      IF (_MessageLevel > E_MessageType.eMessageError)
      THEN
        _stMsg.eType            := E_MessageType.eMessageInfo;
        _stMsg.eSubdevice       := e_Subdevice.Process_LinkedList_Com_DelHead;
        _stMsg.iErrorNumber     := 0;
        _stMsg.sText            := '';
        _stMsg.sText            := concat(_stMsg.sText, TO_STRING(_eState));
        f_MessageSet(_stMsg);
      END_IF
    END_IF
END_CASE
//-----------------------------------------------------------------------------
//-----------------------------------------------------------------------------

ListDelHead                     := _eState;
END_METHOD

METHOD ListDelTail  : e_progress
VAR_INPUT
  Execute           : BOOL;
END_VAR
VAR_INST
  _ListResult       : ST_PROCESS_LIST_RESULT;
  _nErrorId         : UDINT;
  _eState           : E_PROGRESS;
END_VAR
//-----------------------------------------------------------------------------
IF NOT Execute 
THEN 
	_eState                       := E_PROGRESS.PROGRESS_INIT; 
END_IF 
//-----------------------------------------------------------------------------
IF NOT Check() 
THEN 
	ListDelTail                   := E_PROGRESS.PROGRESS_ERROR; 
	RETURN; 
END_IF
//-----------------------------------------------------------------------------
//-----------------------------------------------------------------------------
CASE _eState
OF
  E_PROGRESS.PROGRESS_INIT:
    IF Execute
    THEN
      _nErrorId                 := 0;
      _eState                   := E_PROGRESS.PROGRESS_BUSY;
    END_IF
END_CASE
//-----------------------------------------------------------------------------
//-----------------------------------------------------------------------------
CASE _eState
OF
  E_PROGRESS.PROGRESS_BUSY:
    _eState                     := E_PROGRESS.PROGRESS_PREPARE;
    _ListResult                 := _ItfList.RemoveTailValue();
END_CASE
//-----------------------------------------------------------------------------
//-----------------------------------------------------------------------------
CASE _eState
OF
  E_PROGRESS.PROGRESS_PREPARE:

    IF (_ListResult.wState <> 0)
    THEN
      _eState                   := E_PROGRESS.PROGRESS_ERROR;
      _nErrorId                 := _ListResult.wState;

      _stMsg.eType              := E_MessageType.eMessageError;
      _stMsg.eSubdevice         := e_Subdevice.Process_LinkedList_Com_DelTail;
      _stMsg.iErrorNumber       := _nErrorId;
      _stMsg.sText              := '';
      _stMsg.sText              := concat(_stMsg.sText, TO_STRING(_eState));
      f_MessageSet(_stMsg);

    ELSE
      _eState                   := E_PROGRESS.PROGRESS_DONE;

      IF (_MessageLevel > E_MessageType.eMessageError)
      THEN
        _stMsg.eType            := E_MessageType.eMessageInfo;
        _stMsg.eSubdevice       := e_Subdevice.Process_LinkedList_Com_DelTail;
        _stMsg.iErrorNumber     := 0;
        _stMsg.sText            := '';
        _stMsg.sText            := concat(_stMsg.sText, TO_STRING(_eState));
        f_MessageSet(_stMsg);
      END_IF
    END_IF
END_CASE
//-----------------------------------------------------------------------------
//-----------------------------------------------------------------------------

ListDelTail                     := _eState;
END_METHOD

METHOD ListGetHead  : e_progress
VAR_INPUT
  Execute           : BOOL;
END_VAR
VAR_INST
  _ListResult       : ST_PROCESS_LIST_RESULT;
  _nErrorId         : UDINT;
  _eState           : E_PROGRESS;
END_VAR
//-----------------------------------------------------------------------------
IF NOT Execute 
THEN 
	_eState                         := E_PROGRESS.PROGRESS_INIT; 
END_IF 
//-----------------------------------------------------------------------------
IF NOT Check() 
THEN 
	ListGetHead                     := E_PROGRESS.PROGRESS_ERROR; 
	RETURN; 
END_IF
//-----------------------------------------------------------------------------
//-----------------------------------------------------------------------------
CASE _eState
OF
  E_PROGRESS.PROGRESS_INIT:
    IF Execute
    THEN
      _nErrorId                   := 0;
      _eState                     := E_PROGRESS.PROGRESS_BUSY;
    END_IF
END_CASE
//-----------------------------------------------------------------------------
//-----------------------------------------------------------------------------
CASE _eState
OF
  E_PROGRESS.PROGRESS_BUSY:
    _eState                       := E_PROGRESS.PROGRESS_PREPARE;
    _ListResult                   := _ItfList.GetHead();
END_CASE
//-----------------------------------------------------------------------------
//-----------------------------------------------------------------------------
CASE _eState
OF
  E_PROGRESS.PROGRESS_PREPARE:

    IF (_ListResult.wState <> 0)
    THEN
      _eState                     := E_PROGRESS.PROGRESS_ERROR;
      _nErrorId                   := _ListResult.wState;

      _stMsg.eType                := E_MessageType.eMessageError;
      _stMsg.eSubdevice           := e_Subdevice.Process_LinkedList_Com_GetHead;
      _stMsg.iErrorNumber         := _nErrorId;
      _stMsg.sText                := '';
      _stMsg.sText                := concat(_stMsg.sText, TO_STRING(_eState));
      f_MessageSet(_stMsg);

    ELSE
      _stNodeDataProcess.ProcessData:= _ListResult.stData;
      _stNodeDataOutput             := _stNodeDataProcess;

      _eState                     := E_PROGRESS.PROGRESS_DONE;

      IF (_MessageLevel > E_MessageType.eMessageError)
      THEN
        _stMsg.eType              := E_MessageType.eMessageInfo;
        _stMsg.eSubdevice         := e_Subdevice.Process_LinkedList_Com_GetHead;
        _stMsg.iErrorNumber       := 0;
        _stMsg.sText              := '';
        _stMsg.sText              := concat(_stMsg.sText, TO_STRING(_eState));
        f_MessageSet(_stMsg);
      END_IF
    END_IF
END_CASE
//-----------------------------------------------------------------------------
//-----------------------------------------------------------------------------

ListGetHead                       := _eState;
END_METHOD

METHOD ListGetTail  : e_progress
VAR_INPUT
  Execute           : BOOL;
END_VAR
VAR_INST
  _ListResult       : ST_PROCESS_LIST_RESULT;
  _nErrorId         : UDINT;
  _eState           : E_PROGRESS;
END_VAR
//-----------------------------------------------------------------------------
IF NOT Execute 
THEN 
	_eState                         := E_PROGRESS.PROGRESS_INIT; 
END_IF 
//-----------------------------------------------------------------------------
IF NOT Check() 
THEN 
	ListGetTail                     := E_PROGRESS.PROGRESS_ERROR; 
	RETURN; 
END_IF
//-----------------------------------------------------------------------------
//-----------------------------------------------------------------------------
CASE _eState
OF
  E_PROGRESS.PROGRESS_INIT:
    IF Execute
    THEN
      _nErrorId                   := 0;
      _eState                     := E_PROGRESS.PROGRESS_BUSY;
    END_IF
END_CASE
//-----------------------------------------------------------------------------
//-----------------------------------------------------------------------------
CASE _eState
OF
  E_PROGRESS.PROGRESS_BUSY:
    _eState                       := E_PROGRESS.PROGRESS_PREPARE;
    _ListResult                   := _ItfList.GetTail();
END_CASE
//-----------------------------------------------------------------------------
//-----------------------------------------------------------------------------
CASE _eState
OF
  E_PROGRESS.PROGRESS_PREPARE:

    IF (_ListResult.wState <> 0)
    THEN
      _eState                     := E_PROGRESS.PROGRESS_ERROR;
      _nErrorId                   := _ListResult.wState;

      _stMsg.eType                := E_MessageType.eMessageError;
      _stMsg.eSubdevice           := e_Subdevice.Process_LinkedList_Com_GetTail;
      _stMsg.iErrorNumber         := _nErrorId;
      _stMsg.sText                := '';
      _stMsg.sText                := concat(_stMsg.sText, TO_STRING(_eState));
      f_MessageSet(_stMsg);

    ELSE
      _stNodeDataProcess.ProcessData:= _ListResult.stData;
      _stNodeDataOutput             := _stNodeDataProcess;

      _eState                     := E_PROGRESS.PROGRESS_DONE;

      IF (_MessageLevel > E_MessageType.eMessageError)
      THEN
        _stMsg.eType              := E_MessageType.eMessageInfo;
        _stMsg.eSubdevice         := e_Subdevice.Process_LinkedList_Com_GetTail;
        _stMsg.iErrorNumber       := 0;
        _stMsg.sText              := '';
        _stMsg.sText              := concat(_stMsg.sText, TO_STRING(_eState));
        f_MessageSet(_stMsg);
      END_IF
    END_IF
END_CASE
//-----------------------------------------------------------------------------
//-----------------------------------------------------------------------------

ListGetTail                       := _eState;
END_METHOD

METHOD ListInit  : e_progress
VAR_INPUT
  Execute           : BOOL;
END_VAR
VAR_INST
  _ListResult       : BOOL;

  _nErrorId         : UDINT;
  _eState           : E_PROGRESS;
END_VAR
//-----------------------------------------------------------------------------
IF NOT Execute 
THEN 
	_eState                       := E_PROGRESS.PROGRESS_INIT; 
END_IF 
//-----------------------------------------------------------------------------
IF NOT Check() 
THEN 
	ListInit                      := E_PROGRESS.PROGRESS_ERROR; 
	RETURN; 
END_IF
//-----------------------------------------------------------------------------
//-----------------------------------------------------------------------------
CASE _eState
OF
  E_PROGRESS.PROGRESS_INIT:
    IF Execute
    THEN
      _nErrorId                 := 0;
      _eState                   := E_PROGRESS.PROGRESS_BUSY;
    END_IF
END_CASE
//-----------------------------------------------------------------------------
//-----------------------------------------------------------------------------
CASE _eState
OF
  E_PROGRESS.PROGRESS_BUSY:
    _eState                     := E_PROGRESS.PROGRESS_PREPARE;
    _ListResult                 := _ItfList.InitList();
END_CASE
//-----------------------------------------------------------------------------
//-----------------------------------------------------------------------------
CASE _eState
OF
  E_PROGRESS.PROGRESS_PREPARE:

    IF NOT (_ListResult)
    THEN
      _eState                   := E_PROGRESS.PROGRESS_ERROR;
      _nErrorId                 := 666;

      _stMsg.eType              := E_MessageType.eMessageError;
      _stMsg.eSubdevice         := e_Subdevice.Process_LinkedList_Com_Init;
      _stMsg.iErrorNumber       := _nErrorId;
      _stMsg.sText              := '';
      _stMsg.sText              := concat(_stMsg.sText, TO_STRING(_eState));
      f_MessageSet(_stMsg);

    ELSE
      _eState                   := E_PROGRESS.PROGRESS_DONE;

      IF (_MessageLevel > E_MessageType.eMessageError)
      THEN
        _stMsg.eType            := E_MessageType.eMessageInfo;
        _stMsg.eSubdevice       := e_Subdevice.Process_LinkedList_Com_Init;
        _stMsg.iErrorNumber     := 0;
        _stMsg.sText            := '';
        _stMsg.sText            := concat(_stMsg.sText, TO_STRING(_eState));
        f_MessageSet(_stMsg);
      END_IF
    END_IF
END_CASE
//-----------------------------------------------------------------------------
//-----------------------------------------------------------------------------

ListInit                        := _eState;
END_METHOD

PROPERTY MessageLevel : e_MessageType
GET
MessageLevel := _MessageLevel;
END_GET
SET
_MessageLevel := MessageLevel;
END_SET
END_PROPERTY

PROPERTY NodeDataInput : reference to st_list_node_data
SET
_stNodeDataInput REF= NodeDataInput;
END_SET
END_PROPERTY

PROPERTY NodeDataOutput : reference to st_list_node_data
SET
_stNodeDataOutput REF= NodeDataOutput;
END_SET
END_PROPERTY

PROPERTY State : REFERENCE TO ST_LIST_STATE
SET
_stState ref= State;
END_SET
END_PROPERTY

END_FUNCTION_BLOCK

// ---- XTS_TRANSPORT/MAIN_XTS.TcPOU
//---------------------------------------------------------------------------------------------------------------
//
//  HAUD 2026.07.25
//  - refactoring update
//    - folder structure accommodates PLC_MOTION_LAYER MSG declarations
//      - This shall help to have both projects merged into one codebase
//        - merging this into a single codebase is up to you, 
//          the machines I do are vastly different in that regard
//          I merge what I need for an implementation / example
//
//    - PRGs are in their corresponding folders
//      - MAIN_XTS --> [XTS]
//      - MAIN_APP --> [APPLICATION]
//
//    - Manage the call tree when merging --> PlcTask.TcTTO
//
//---------------------------------------------------------------------------------------------------------------
//
//  HAUD 2026.07.24
//  - message system refactoring
//    - XTS_TRANSPORT_LAYER and PLC_MOTION_LAYER merged devices
//      - GVL naming conflict resolved
//---------------------------------------------------------------------------------------------------------------
//
//  HAUD 2026.04.23
//  - fb_Xpu
//    - .Init() initialisation sequence with explicit init of all local instances
//    - .GetPartModule added, gets all Tc3_XTS_Utility.I_TcIoXtsPartModule 
// 
//  - MAPPING
//    - MOVER_SELECTOR and MOVER_MAPPING compile defines are mutually exclusive.
//    - switching memcpy destinations/sources according to compile define
//
//  - I_XtsTransport_Xpu
//    - you might need this interface to access methods for passing along the XTS_Utility interfaces
//
// 
//---------------------------------------------------------------------------------------------------------------
//
//  HAUD 2026.03.15
//  - refactoring of the constants
//  - I never really used the parameter list anyway 
//
//  - XTS Utility lib parameter and project constants now reside in:
//    GVL_XTS_CONSTANTS
//
//  - addition of MAIN_APP (also see call tree)
//    - this might be a point of entry for you
//    - advanced transport logic may live here
//    - Beware the Collectors, they need instances to be really useful
//
//---------------------------------------------------------------------------------------------------------------
//
//  HAUD 2026.02.11
//  - transport layer new member:
//    - MoverSelector
//      - Cyclic movement execution class
//      - mapping unions available
//      - Mover selection (one mover at a time)
//      - composition using I_XtsTransport_Mover
//
//
//---------------------------------------------------------------------------------------------------------------
//
//  HAUD 2025.12.04
//
//  - XTS_TRANSPORT_LAYER
//  - transport layer members:
//    - MessageData
//      - ABSTRACT base class
//        - cyclic wrapper
//
//      - device driven message list implementation
//        - e_Device.Metrics: message list dedicated for performance logs
//
//      - new e_MessageType
//        -  eMessageBatch: may be used for performance metric messages
//
//    - CaGroup
//      - access to Group functions
//
//    - Mover
//      - Base class
//        - cyclic wrapper
//
//      - access to MC and CA motion functions
//
//    - Xpu (ProcessingUnit)
//      - Base class
//        - cyclic wrapper
//
//      - access to TcCOM Objects in Environment
//
//    - Transport Control Unit
//      - coordinates members to get XTS in defined states
//
//    - Xts Stations
//      - ABSTRACT base class
//        - used via inheritance
//
//      - handshakes with extern control for mover transport
//
//  - global datafields for mrmbers in GVL_XTS namespace
//  - global interface datafields for use in members
//  - structures are assigned by reference for every member
//
//---------------------------------------------------------------------------------------------------------------
// HAUD 2025 08 29
//
//    XTS_TRANSPORT_LAYER project
//    
//    MIT License
//    
//    Copyright (c) 2025 HAUD
//    
//    Permission is hereby granted, free of charge, to any person obtaining a copy
//    of this software and associated documentation files (the "Software"), to deal
//    in the Software without restriction, including without limitation the rights
//    to use, copy, modify, merge, publish, distribute, sublicense, and/or sell
//    copies of the Software, and to permit persons to whom the Software is
//    furnished to do so, subject to the following conditions:
//    
//    The above copyright notice and this permission notice shall be included in all
//    copies or substantial portions of the Software.
//    
//    THE SOFTWARE IS PROVIDED "AS IS", WITHOUT WARRANTY OF ANY KIND, EXPRESS OR
//    IMPLIED, INCLUDING BUT NOT LIMITED TO THE WARRANTIES OF MERCHANTABILITY,
//    FITNESS FOR A PARTICULAR PURPOSE AND NONINFRINGEMENT. IN NO EVENT SHALL THE
//    AUTHORS OR COPYRIGHT HOLDERS BE LIABLE FOR ANY CLAIM, DAMAGES OR OTHER
//    LIABILITY, WHETHER IN AN ACTION OF CONTRACT, TORT OR OTHERWISE, ARISING FROM,
//    OUT OF OR IN CONNECTION WITH THE SOFTWARE OR THE USE OR OTHER DEALINGS IN THE
//    SOFTWARE.
//---------------------------------------------------------------------------------------------------------------
PROGRAM MAIN_XTS
VAR
  //-------------------------------------------------------------------------------------------------------------
  //  MAIN - important members
  //-------------------------------------------------------------------------------------------------------------
  eInit                   : E_PROGRESS; // startup states
  eInitError              : E_PROGRESS; // startup error state: NOT_EXIST --> NO_ERROR

  nStation,
	nMover                  : UINT;
  //-------------------------------------------------------------------------------------------------------------
  //-------------------------------------------------------------------------------------------------------------
  // default initialization data
  //-------------------------------------------------------------------------------------------------------------
  nStn                    : UINT;               // startup default data, do not delete
  rInitVelo               : REAL :=     500.0;  // default data, use your own in a real machine!
  rInitGap                : REAL :=     100.0;  // default data, use your own in a real machine!
  rInitAcc                : REAL :=  10_000.0;  // default data, use your own in a real machine!
  rInitJerk               : REAL := 100_000.0;  // default data, use your own in a real machine!
  //-------------------------------------------------------------------------------------------------------------
  //-------------------------------------------------------------------------------------------------------------
  // message data used here in MAIN (init state machine etc.)
  //-------------------------------------------------------------------------------------------------------------
  stMsg                   : ST_Message;
  eMsgState               : e_message_state;
  eMsgProgress            : E_PROGRESS;
  eMtrState               : e_message_state;
  eMtrProgress            : E_PROGRESS;
  //-------------------------------------------------------------------------------------------------------------
  //-------------------------------------------------------------------------------------------------------------
  // visualisations - the helper visus depend on these
  //                - the helper visus are just that
  //-------------------------------------------------------------------------------------------------------------
  nMoverSelected,
  nStationSelected,
  nStationParameter       : UINT;

  sStationText            : STRING(30);
  stXpuStrings            : ST_XPU_STRINGS;

  eTransportState         : E_XTS_TRANSPORT_STATE;
  eTransportResult        : E_PROGRESS;

  eXpuState               : E_XPU_STATE;
  eXpuResult              : E_PROGRESS;
  eXpuCheck               : E_XPU_CHECK;

  eSelectorState,
  eMoverState             : E_MOVER_STATE;

  eSelectorResult,
  eMoverResult            : E_PROGRESS;

  sSelectorState,
  sSelectorResult,
  sCaGroupState,
  sTransportState,
  sTransportCheck,
  sTransportResult,
  sMoverState,
  sMoverResult,
  sStationState,
  sStationStateMask,
  sStationCtrlMask        : STRING;

  bStationEnable,
  bStationEnter,
  bStationStart,
  bStationDone,
  bStationOut,
  bStationGone            : BOOL;

  tStationSelectedQueue   : ARRAY[1..MAX_LIST_NODES] OF ST_STATION_MOVER_DATA;
  //-------------------------------------------------------------------------------------------------------------
  tIdleWriteMotion        : TIME := T#5S;
  tIdleWriteMetric        : TIME := T#5S;
  tonIdleWriteMotion      : Tc2_Standard.TON;
  tonIdleWriteMetric      : Tc2_Standard.TON;
  //-------------------------------------------------------------------------------------------------------------
END_VAR

//############################################################################
// Local time; used for timestamps
//############################################################################
GVL_MSG_XTS.fbLocalTime();
GVL_MSG_XTS.sLocalTime                              := GVL_MSG_XTS.fbLocalTime.LocalTimeString;
GVL_MSG_XTS.dtLocalTime                             := GVL_MSG_XTS.fbLocalTime.LocalTime;
//############################################################################
//############################################################################
// 	example for init sequence
//############################################################################	
CASE eInit
OF
  E_PROGRESS.PROGRESS_INVALID:
    // In the beginning there was no error...
    eInitError                                  := E_PROGRESS.PROGRESS_NOT_EXIST;
    //---------------------------------------------------------------------------
    // where are the stations?
    // TODO: after importing this project into your XTS TwinCAT solution
    //       setup of Station parameters is required.
    //---------------------------------------------------------------------------
    // default initialization, please leave this in here
    DefaultStationParameters();        
    //---------------------------------------------------------------------------
    //---------------------------------------------------------------------------
    // where to start?
    // fb_TransportUnit is connected StationStartIndex and StationStart
    //
    // TODO: after importing this project into your XTS TwinCAT solution
    //       setup of StartStation parameters is up to you to decide.
    //---------------------------------------------------------------------------
    GVL_XTS.StationStartIndex                   := 1; // this index is yours to change, fbTransportUnit is connected to it
    GVL_XTS.StationStart                        := GVL_XTS.StationParameter[GVL_XTS.StationStartIndex]; // put in here any plausible data you like
    //---------------------------------------------------------------------------

    eInit                                       := E_PROGRESS.PROGRESS_BUSY;
    // clear command interface
    GVL_XTS.XpuCtrl.Cmd                         := E_XPU_CTRL.XTS_CMD_NULL;
    GVL_MSG_XTS.TransportMessageCtrl.Cmd            := E_MESSAGE_CTRL.MSG_CTRL_NULL;
    GVL_MSG_XTS.MetricsMessageCtrl.Cmd              := E_MESSAGE_CTRL.MSG_CTRL_NULL;

    // set detailed message levvel for startup
    GVL_MSG_XTS.MessageLevelXpu                     := E_MessageType.eMessageVerbose; //GVL_MSG.MessageLevel;
    GVL_XTS.CaGroup.MessageLevel                := E_MessageType.eMessageVerbose; //GVL_MSG.MessageLevel;
    GVL_XTS.XtsTransport.MessageLevel           := E_MessageType.eMessageVerbose; //GVL_MSG.MessageLevel;

    FOR nStation := 1 TO MAX_STATION
    DO
      GVL_MSG_XTS.MessageLevelStations[nStation]    := E_MessageType.eMessageVerbose; //GVL_MSG.MessageLevel;
    END_FOR
    FOR nMover := 1 TO MAX_MOVER
    DO
      GVL_MSG_XTS.MessageLevelMovers[nMover]        := E_MessageType.eMessageVerbose; //GVL_MSG.MessageLevel;
    END_FOR
    
  //-----------------------------------------------------------------------------
  //-----------------------------------------------------------------------------
  E_PROGRESS.PROGRESS_BUSY:         // init Xpu, ProcessingUnit, MotorModules
    eInit                                       := E_PROGRESS.PROGRESS_PREPARE;
    GVL_MSG_XTS.TransportMessageCtrl.Cmd            := E_MESSAGE_CTRL.MSG_CTRL_INIT;
    GVL_MSG_XTS.MetricsMessageCtrl.Cmd              := E_MESSAGE_CTRL.MSG_CTRL_INIT;


  //-----------------------------------------------------------------------------
  //-----------------------------------------------------------------------------
  E_PROGRESS.PROGRESS_PREPARE:      // wait for init to be done
    GVL_XTS.XpuCtrl.Cmd                         := E_XPU_CTRL.XTS_CMD_INIT;
    IF (GVL_XTS.XpuState.State      = E_XPU_STATE.XTS_INIT + E_PROGRESS.PROGRESS_ERROR)
    THEN
      stMsg.eType                               := E_MessageType.eMessageInfo;
      stMsg.eDevice                             := e_Device.Device_Main;
      stMsg.eSubdevice                          := e_Subdevice.MainInit;
      stMsg.iErrorNumber                        := GVL_XTS.XpuState.Check;
      stMsg.sText                               := concat('MAIN.eInit Error: ', TO_STRING(MAIN_XTS.eInit));
      stMsg.sText                               := concat(stMsg.sText , ': ');
      stMsg.sText                               := concat(stMsg.sText, 'XpuState.Check: ');
      stMsg.sText                               := concat(stMsg.sText, TO_STRING(GVL_XTS.XpuState.Check));
      f_MessageSet(stMsg);

      eInitError                                := eInit;
      eInit                                     := E_PROGRESS.PROGRESS_ERROR;

    ELSIF (GVL_XTS.XpuState.State   = E_XPU_STATE.XTS_INIT + E_PROGRESS.PROGRESS_DONE)
    THEN
      eInit                                     := E_PROGRESS.PROGRESS_STARTUP;
      GVL_XTS.XpuCtrl.Cmd                       := E_XPU_CTRL.XTS_IDLE;
    END_IF

  //-----------------------------------------------------------------------------
  //-----------------------------------------------------------------------------
  E_PROGRESS.PROGRESS_STARTUP:
    CASE GVL_XTS.XpuState.Check
    OF
      E_XPU_CHECK.MOVER_ID_SIMULATION,
      E_XPU_CHECK.MOVER_ID_DETECTION_VALID:
        IF (GVL_XTS.XpuState.State = E_XPU_STATE.XTS_IDLE + E_PROGRESS.PROGRESS_WORKING)
        THEN
          eInit                                     := E_PROGRESS.PROGRESS_CHECK;
        END_IF
    END_CASE
  //-----------------------------------------------------------------------------
  //-----------------------------------------------------------------------------
  E_PROGRESS.PROGRESS_CHECK:
    eInit                                       := E_PROGRESS.PROGRESS_OCCUPIED;

  //-----------------------------------------------------------------------------
  //-----------------------------------------------------------------------------
  E_PROGRESS.PROGRESS_OCCUPIED:
    //---------------------------------------------------------------------------
    // how many nests to start with?
    // - this is for you to decide and me to secure, 
    //    so leave the initialisation as it is
    //
    // TODO: after importing this project into your XTS TwinCAT solution
    //       setup of StartStation NestMask configuration is up to you to decide.
    //---------------------------------------------------------------------------
    IF (GVL_XTS.XtsTransport.StationStartIndex > 0) AND
       (GVL_XTS.XtsTransport.StationStartIndex < MAX_STATION+1)
    THEN
      GVL_XTS.StationStart.nConfiguredStopCount := GVL_XTS.StationParameter[GVL_XTS.XtsTransport.StationStartIndex].nConfiguredStopCount;
    END_IF
    eInit                                       := E_PROGRESS.PROGRESS_WORKING;

  //-----------------------------------------------------------------------------
  //-----------------------------------------------------------------------------
  E_PROGRESS.PROGRESS_WORKING:
    GVL_MSG_XTS.TransportMessageCtrl.Cmd            := E_MESSAGE_CTRL.MSG_CTRL_WRITE;
    eInit                                       := E_PROGRESS.PROGRESS_DONE;

    stMsg.eType                                 := E_MessageType.eMessageInfo;
    stMsg.eDevice                               := e_Device.Device_Main;
    stMsg.eSubdevice                            := e_Subdevice.MainInit;
    stMsg.iErrorNumber                          := GVL_XTS.XpuState.Check;
    stMsg.sText                                 := concat('MAIN.eInit Done: ', TO_STRING(MAIN_XTS.eInit));
    stMsg.sText                                 := concat(stMsg.sText , ': ');
    stMsg.sText                                 := concat(stMsg.sText, 'XpuState.Check: ');
    stMsg.sText                                 := concat(stMsg.sText, TO_STRING(GVL_XTS.XpuState.Check));
    f_MessageSet(stMsg);

    //---------------------------------------------------------------------------
END_CASE
//############################################################################
//############################################################################
// 	/XTS Transport Unit
//############################################################################
//  - main control function block for transport layer
//  - requires access to member controls
//    - Xpu
//    - CaGroup
//    - Mover
//    - Station Control
//    - Station LinkedList Interface
//############################################################################
//
// cyclic call
GVL_XTS.XtsTransport();

// main control
GVL_XTS.XtsTransport.Ctrl                       REF= GVL_XTS.XtsTransportCtrl;   // main control
GVL_XTS.XtsTransport.State                      REF= GVL_XTS.XtsTransportState;  // main state
                                        
// member controls                      
GVL_XTS.XtsTransport.XpuCtrl                    REF= GVL_XTS.XpuCtrl;
GVL_XTS.XtsTransport.XpuState                   REF= GVL_XTS.XpuState;
GVL_XTS.XtsTransport.XpuInfo                    REF= GVL_XTS.XpuInfo;
                                        
GVL_XTS.XtsTransport.GroupItf                   :=   GVL_XTS.CaGroupItf;
GVL_XTS.XtsTransport.GroupInfo                  REF= GVL_XTS.CaGroupInfo;
                                        
GVL_XTS.XtsTransport.MoverItf                   REF= GVL_XTS.MoverItf;
GVL_XTS.XtsTransport.MoverInfo                  REF= GVL_XTS.MoverInfo;
GVL_XTS.XtsTransport.MoverLastPosition          REF= GVL_XTS.LastPosition;
GVL_XTS.XtsTransport.MoverLastGap               REF= GVL_XTS.LastGap;

GVL_XTS.XtsTransport.StationStartIndex          :=   GVL_XTS.StationStartIndex;                                        
GVL_XTS.XtsTransport.StationStart               REF= GVL_XTS.StationStart;      // start position for E_XTS_TRANSPORT_CTRL.CMD_TRANSPORT_START
GVL_XTS.XtsTransport.StationCtrlItf             REF= GVL_XTS.StationCtrlItf;    // station interfaces are required for accessing station methods
GVL_XTS.XtsTransport.StationListsItf            REF= GVL_XTS.StationListItf;    // list interface is required for access to linked list methods
GVL_XTS.XtsTransport.StationControl             REF= GVL_XTS.StationCtrl;
GVL_XTS.XtsTransport.StationState               REF= GVL_XTS.StationState;
//############################################################################
// 	XTS Transport Unit/
//############################################################################
//############################################################################
//############################################################################
// 	/XTS Stations
//############################################################################	
FOR nStation := 1 TO MAX_STATION
DO
  // epimetheus assembles the body
  GVL_XTS.StationListItf[nStation]              := GVL_XTS.StationList[nStation];   // interfaces for list methods
  GVL_XTS.StationCtrlItf[nStation]              := GVL_XTS.Station[nStation];       // interfaces for station methods

  CASE GVL_XTS.StationParameter[nStation].eType
  OF
    //-----------------------------------------------------------------------------
    E_STATION_TYPE.STATION_PROCESS:
      GVL_XTS.Station[nStation].MessageLevel    := GVL_MSG_XTS.MessageLevelStations[nStation];

      GVL_XTS.Station[nStation].StationId       := nStation;  // Know Thyself!

    
      GVL_XTS.Station[nStation].Ctrl            REF= GVL_XTS.StationCtrl;           // station ctrl from extern
      GVL_XTS.Station[nStation].State           REF= GVL_XTS.StationState;          // station state to extern
    
      GVL_XTS.Station[nStation].ItfStations     REF= GVL_XTS.StationListItf;        // give every station all list interfaces for writing mover tickets
      GVL_XTS.Station[nStation].ItfMover        REF= GVL_XTS.MoverItf;              // give every station all mover interfaces for movement in / out of station
      GVL_XTS.Station[nStation].Mover           REF= GVL_XTS.AxisRefMover;          // AXIS_REF to read infos from
      GVL_XTS.Station[nStation].MoverOffset     REF= GVL_XTS.PositionOffset;        // static offsets for all stations, all movers, all stop positions
    
      GVL_XTS.Station[nStation].StationParameter  REF= GVL_XTS.StationParameter;// give every station all station parameters for sending to WaitPos of target station
    
      // cyclic call
      GVL_XTS.Station[nStation].Cycle();                                        // cycle for handshaking with extern
    
      // Queue data for each station
      GVL_XTS.StationQueue[nStation]            := GVL_XTS.StationListItf[nStation].Data;


    //-----------------------------------------------------------------------------
    E_STATION_TYPE.STATION_GEAR_IN_POS:
      GVL_XTS.StationGearIn[nStation].MessageLevel:= GVL_MSG_XTS.MessageLevelStations[nStation];

      GVL_XTS.Station[nStation].StationId         := nStation;  // Know Thyself!
    
      GVL_XTS.StationGearIn[nStation].Ctrl        REF= GVL_XTS.StationCtrl;           // station ctrl from extern
      GVL_XTS.StationGearIn[nStation].State       REF= GVL_XTS.StationState;          // station state to extern
    
      GVL_XTS.StationGearIn[nStation].ItfStations REF= GVL_XTS.StationListItf;        // give every station all list interfaces for writing mover tickets
      GVL_XTS.StationGearIn[nStation].ItfMover    REF= GVL_XTS.MoverItf;              // give every station all mover interfaces for movement in / out of station
      GVL_XTS.StationGearIn[nStation].Mover       REF= GVL_XTS.AxisRefMover;          // AXIS_REF to read infos from
      GVL_XTS.StationGearIn[nStation].MoverOffset REF= GVL_XTS.PositionOffset;        // static offsets for all stations, all movers, all stop positions
    
    
      GVL_XTS.StationGearIn[nStation].StationParameter  REF= GVL_XTS.StationParameter;// give every station all station parameters for sending to WaitPos of target station
    
      // cyclic call
      GVL_XTS.StationGearIn[nStation].Cycle();                                        // cycle for handshaking with extern
    
      // Queue data for each station
      GVL_XTS.StationQueue[nStation]            := GVL_XTS.StationListItf[nStation].Data;
  ELSE
      //---------------------------------------------------------------------------------
      // no valid station type --> no identity
      //---------------------------------------------------------------------------------
      GVL_XTS.Station[nStation].StationId       := 0; // I am no one
      //---------------------------------------------------------------------------------
  END_CASE
END_FOR
//############################################################################
// 	XTS Stations/
//############################################################################	
//############################################################################
//############################################################################
// 	/XPU environment
//############################################################################	
GVL_XTS.Xpu.XpuInstance                         :=   1;
GVL_XTS.Xpu.MessageLevel                        :=   GVL_MSG_XTS.MessageLevelXpu;

GVL_XTS.Xpu.Ctrl                                REF= GVL_XTS.XpuCtrl;
GVL_XTS.Xpu.State                               REF= GVL_XTS.XpuState;
GVL_XTS.Xpu.XpuModuleInfoData                   REF= GVL_XTS.XpuModules;

GVL_XTS.Xpu.CaGroupOID                          :=   GVL_XTS.CaGroup.GroupInfo.CaGroupOID;

// cyclic call                                
GVL_XTS.Xpu();                                
GVL_XTS.XpuInfo                                 :=   GVL_XTS.Xpu.XpuInfo;
//############################################################################
// 	XPU environment/
//############################################################################	
//############################################################################
//############################################################################	
// 	/CA-Group Class
//############################################################################
// message device identifier
GVL_XTS.CaGroup.MessageDeviceIndex              :=   e_Device.CaGroup + 1;	
// assignment
GVL_XTS.CaGroup.AxisRef                         REF= GVL_XTS.AxisRefMover;
// Interface to Mover methods
GVL_XTS.CaGroup.MoverItf                        REF= GVL_XTS.MoverItf; 
GVL_XTS.CaGroup.GroupRef                        REF= GVL_XTS.CaGroupRef;
GVL_XTS.CaGroup.XpuInfo                         REF= GVL_XTS.XpuInfo;
// cyclic call
GVL_XTS.CaGroup.InfoCycle(TRUE);                // read group status
// InfoData from group
GVL_XTS.CaGroupInfo                             :=   GVL_XTS.CaGroup.GroupInfo;
// Interface of CaGroup
GVL_XTS.CaGroupItf                              :=   GVL_XTS.CaGroup;
//############################################################################	
// 	CA-Group Class/
//############################################################################
//############################################################################
//############################################################################
//  /Mover Class	
//############################################################################	
FOR nMover := 1 TO MAX_MOVER
DO
  GVL_XTS.Mover[nMover].MoverId                 :=   nMover;
  GVL_XTS.Mover[nMover].RailLength              :=   GVL_XTS.Xpu.RailLength;  // mover needs RailLength, in order to calc absolute position from modulo input
  GVL_XTS.Mover[nMover].MessageLevel            :=   GVL_MSG_XTS.MessageLevelMovers[nMover];

  GVL_XTS.Mover[nMover].Ctrl                    REF= GVL_XTS.MoverCtrl;       // mover control from extern
  GVL_XTS.Mover[nMover].State                   REF= GVL_XTS.MoverState;      // mover state to extern

  GVL_XTS.Mover[nMover].MoveData                REF= GVL_XTS.MoveData;        // dyn constraints for extern to write
  GVL_XTS.Mover[nMover].GearData                REF= GVL_XTS.GearData;        // GearIn/GearInPosCa data fro extern to write

  // assignment
  GVL_XTS.Mover[nMover].Mover                   REF= GVL_XTS.AxisRefMover[nMover];  // axis reference to Mover function block
  GVL_XTS.Mover[nMover].LastGap                 REF= GVL_XTS.LastGap[nMover];       // reference to last used gap value datafield
  GVL_XTS.Mover[nMover].LastPosition            REF= GVL_XTS.LastPosition[nMover];  // reference to last position datafield

  GVL_XTS.Mover[nMover].MoverInfo		            REF= GVL_XTS.MoverInfo[nMover];     // refernence to mover info data (ActPos, SetPos, ...)

  GVL_XTS.MoverItf[nMover]                      :=   GVL_XTS.Mover[nMover];

  // cyclic call
  GVL_XTS.Mover[nMover].Cycle();                // call AXIS_REF()
  GVL_XTS.Mover[nMover]();                      // call Ctrl/State
END_FOR
//############################################################################
//  Mover Class/	
//############################################################################	
//############################################################################
//############################################################################
//  /Mover Selector	
//############################################################################
GVL_XTS.MoverSelector.Ctrl                      REF= GVL_XTS.MoverSelectorCtrl;
GVL_XTS.MoverSelector.State                     REF= GVL_XTS.MoverSelectorState;
GVL_XTS.MoverSelector.AxisRef                   REF= GVL_XTS.AxisRefMover;
GVL_XTS.MoverSelector.Info                      REF= GVL_XTS.MoverInfo;
GVL_XTS.MoverSelector.ItfMover                  REF= GVL_XTS.MoverItf;

GVL_XTS.MoverSelector();
//############################################################################
//  Mover Selector/	
//############################################################################	
//############################################################################
//############################################################################
//  /logging
//    - all life is problem solving
//############################################################################
GVL_MSG_XTS.TransportMessageData.Ctrl               REF= GVL_MSG_XTS.TransportMessageCtrl;
GVL_MSG_XTS.TransportMessageData.State              REF= GVL_MSG_XTS.TransportMessageState;
GVL_MSG_XTS.TransportMessageData.MessageIndex       REF= GVL_MSG_XTS.MessageTransportIndex;
GVL_MSG_XTS.TransportMessageData.ErrorIndex         REF= GVL_MSG_XTS.MessageTransportError;
GVL_MSG_XTS.TransportMessageData.DirRoot            :=   ADR(GVL_MSG_XTS.LOG_DIR);
GVL_MSG_XTS.TransportMessageData.FileRoot           :=   ADR(GVL_MSG_XTS.LOG_FILE);
GVL_MSG_XTS.TransportMessageData.MsgList            :=   ADR(GVL_MSG_XTS.TransportMessages);
GVL_MSG_XTS.TransportMessageData.LocalTime          :=   ADR(GVL_MSG_XTS.dtLocalTime);
GVL_MSG_XTS.TransportMessageData();
eMsgState                                       :=   f_GetState   (GVL_MSG_XTS.TransportMessageState.State);
eMsgProgress                                    :=   f_GetProgress(GVL_MSG_XTS.TransportMessageState.State);

CASE eMsgState
OF
  E_MESSAGE_STATE.MSG_STATE_NULL:
    CASE eMsgProgress
    OF
      E_PROGRESS.PROGRESS_INVALID,
      E_PROGRESS.PROGRESS_DONE:
        IF (GVL_MSG_XTS.MessageTransportIndex > GVL_MSG_XTS.MAX_MESSAGE/100) OR
           (GVL_MSG_XTS.MessageTransportError > 0)
        THEN
          GVL_MSG_XTS.TransportMessageCtrl.Cmd      := E_MESSAGE_CTRL.MSG_CTRL_WRITE;
        ELSE
          tonIdleWriteMotion(IN := TRUE, PT:= tIdleWriteMotion);
          IF (tonIdleWriteMotion.Q)
          THEN
            GVL_MSG_XTS.TransportMessageCtrl.Cmd    := E_MESSAGE_CTRL.MSG_CTRL_WRITE;
          END_IF
        END_IF
    END_CASE

  E_MESSAGE_STATE.MSG_STATE_WRITE:
    CASE eMsgProgress
    OF
      E_PROGRESS.PROGRESS_ERROR,
      E_PROGRESS.PROGRESS_DONE:
          tonIdleWriteMotion(IN := FALSE, PT:= tIdleWriteMotion);
        GVL_MSG_XTS.TransportMessageCtrl.Cmd        := E_MESSAGE_CTRL.MSG_CTRL_NULL;
    END_CASE

ELSE
    CASE eMsgProgress
    OF
      E_PROGRESS.PROGRESS_DONE:
        GVL_MSG_XTS.TransportMessageCtrl.Cmd        := E_MESSAGE_CTRL.MSG_CTRL_NULL;
    END_CASE
END_CASE
//############################################################################
//  logging/
//############################################################################
//############################################################################
//############################################################################
//  /Transport Metrics
//############################################################################
GVL_MSG_XTS.MetricsMessageData.Ctrl                 REF= GVL_MSG_XTS.MetricsMessageCtrl;
GVL_MSG_XTS.MetricsMessageData.State                REF= GVL_MSG_XTS.MetricsMessageState;

GVL_MSG_XTS.MetricsMessageData.MessageIndex         REF= GVL_MSG_XTS.MessageMetricsIndex;
GVL_MSG_XTS.MetricsMessageData.ErrorIndex           REF= GVL_MSG_XTS.MessageMetricsError;

GVL_MSG_XTS.MetricsMessageData.DirRoot              :=   ADR(GVL_MSG_XTS.LOG_DIR);
GVL_MSG_XTS.MetricsMessageData.FileRoot             :=   ADR(GVL_MSG_XTS.LOG_FILE_METRIC);

GVL_MSG_XTS.MetricsMessageData.MsgList              :=   ADR(GVL_MSG_XTS.MetricsMessages);
GVL_MSG_XTS.MetricsMessageData.LocalTime            :=   ADR(GVL_MSG_XTS.dtLocalTime);

GVL_MSG_XTS.MetricsMessageData();

eMtrState                                       := f_GetState   (GVL_MSG_XTS.MetricsMessageState.State);
eMtrProgress                                    := f_GetProgress(GVL_MSG_XTS.MetricsMessageState.State);

CASE eMtrState
OF
  E_MESSAGE_STATE.MSG_STATE_NULL:
    CASE eMtrProgress
    OF
      E_PROGRESS.PROGRESS_INVALID:
        IF (GVL_MSG_XTS.MessageMetricsIndex > GVL_MSG_XTS.MAX_MESSAGE/100) OR
           (GVL_MSG_XTS.MessageMetricsError > 0)
        THEN
          GVL_MSG_XTS.MetricsMessageCtrl.Cmd        := E_MESSAGE_CTRL.MSG_CTRL_WRITE;
        ELSE
          tonIdleWriteMetric(IN := TRUE, PT:= tIdleWriteMetric);
          IF (tonIdleWriteMetric.Q)
          THEN
            GVL_MSG_XTS.MetricsMessageCtrl.Cmd      := E_MESSAGE_CTRL.MSG_CTRL_WRITE;
          END_IF
        END_IF
    END_CASE

  E_MESSAGE_STATE.MSG_STATE_WRITE:
    CASE eMtrProgress
    OF
      E_PROGRESS.PROGRESS_ERROR,
      E_PROGRESS.PROGRESS_DONE:
        tonIdleWriteMetric(IN := FALSE, PT:= tIdleWriteMetric);
        GVL_MSG_XTS.MetricsMessageCtrl.Cmd          := E_MESSAGE_CTRL.MSG_CTRL_NULL;
    END_CASE
ELSE
    CASE eMtrProgress
    OF
      E_PROGRESS.PROGRESS_DONE:
        GVL_MSG_XTS.MetricsMessageCtrl.Cmd          := E_MESSAGE_CTRL.MSG_CTRL_NULL;
    END_CASE
END_CASE
//############################################################################
//  Transport Metrics/
//############################################################################
//############################################################################
//############################################################################
//  /Visualization data	
//############################################################################
VisualizationData();
//############################################################################
//  Visualization data/	
//############################################################################

ACTION DefaultStationParameters:
//---------------------------------------------------------------------------------------
//---------------------------------------------------------------------------------------
//
//  Default Station dynamics 
//  - we do not want an array full of nothing 
//  - better have something
//  - leave this initialisation as it is, 
//  - go to MAIN_APP to configure the global datafields
//
//---------------------------------------------------------------------------------------
//---------------------------------------------------------------------------------------
FOR nStn := 1 TO MAX_STATION
DO
  GVL_XTS.StationParameter[nStn].eType               :=   E_STATION_TYPE.INVALID; // make it valid in your configuration
  GVL_XTS.StationParameter[nStn].sText               :=   concat('DEaF_STATION_', TO_STRING(nStn));

  GVL_XTS.StationParameter[nStn].rPosWait            :=   TO_REAL(ABS(GVL_XTS.XpuInfo.rRailLength - nStn*10.0));
  GVL_XTS.StationParameter[nStn].rGap                :=   rInitGap;
  GVL_XTS.StationParameter[nStn].rVelo               :=   rInitVelo;
  GVL_XTS.StationParameter[nStn].rAccDec             :=   rInitAcc;
  GVL_XTS.StationParameter[nStn].rJerk               :=   rInitJerk;
END_FOR
//---------------------------------------------------------------------------------------
//---------------------------------------------------------------------------------------
END_ACTION

ACTION VisualizationData:
//############################################################################
//############################################################################
// Visualization data	
//############################################################################
// get enumerations from XPU for visu:	
eTransportState                       := f_GetState   (GVL_XTS.XtsTransportState.State);
eTransportResult                      := f_GetProgress(GVL_XTS.XtsTransportState.State);

eXpuState                             := f_GetState   (GVL_XTS.XtsTransportState.XpuState.State);
eXpuResult                            := f_GetProgress(GVL_XTS.XtsTransportState.XpuState.State);

eXpuCheck                             := GVL_XTS.XtsTransportState.XpuState.Check;

// display xpu state and result in visu
// get strings and info
sCaGroupState                         := TO_STRING(GVL_XTS.XtsTransportState.GroupInfo.CaGroupState);

sTransportState                       := TO_STRING(eTransportState);
sTransportCheck                       := TO_STRING(GVL_XTS.XtsTransportState.Check);
sTransportResult                      := TO_STRING(eTransportResult);

stXpuStrings.sXpuState                := TO_STRING(eXpuState);
stXpuStrings.sXpuResult               := TO_STRING(eXpuResult);
stXpuStrings.sXpuCyclicCheck          := TO_STRING(eXpuCheck);

stXpuStrings.sXpuOpMode               := GVL_XTS.Xpu.OpModeToString();
stXpuStrings.sXpuMoverId_DetectionMode:= GVL_XTS.Xpu.IdDetectionModeToString();
stXpuStrings.sXpuMoverPosAssignement  := GVL_XTS.Xpu.MoverPositionAssignementToString();

nMoverSelected                        := SEL((nMoverSelected<1), nMoverSelected, 1);
nMoverSelected                        := SEL((nMoverSelected>MAX_MOVER), nMoverSelected, MAX_MOVER);

nStationSelected                      := SEL((nStationSelected<1), nStationSelected, 1);
nStationSelected                      := SEL((nStationSelected>MAX_STATION), nStationSelected, MAX_STATION);

bStationEnable                        := SEL((GVL_XTS.StationCtrl[nStationSelected].Cmd = E_STATION_CTRL.STATION_ENABLE),        FALSE, TRUE);
bStationEnter                         := SEL((GVL_XTS.StationCtrl[nStationSelected].Cmd = E_STATION_CTRL.STATION_MOVER_ENTER),   FALSE, TRUE);
bStationStart                         := SEL((GVL_XTS.StationCtrl[nStationSelected].Cmd = E_STATION_CTRL.STATION_PROCESS_START), FALSE, TRUE);
bStationDone                          := SEL((GVL_XTS.StationCtrl[nStationSelected].Cmd = E_STATION_CTRL.STATION_PROCESS_DONE),  FALSE, TRUE);
bStationOut                           := SEL((GVL_XTS.StationCtrl[nStationSelected].Cmd = E_STATION_CTRL.STATION_MOVER_OUT),     FALSE, TRUE);
bStationGone                          := SEL((GVL_XTS.StationCtrl[nStationSelected].Cmd = E_STATION_CTRL.STATION_MOVER_GONE),    FALSE, TRUE);

eMoverState                           := f_GetState   (GVL_XTS.MoverState[nMoverSelected].State);
eMoverResult                          := f_GetProgress(GVL_XTS.MoverState[nMoverSelected].State);

sMoverState                           := TO_STRING(eMoverState);
sMoverResult                          := TO_STRING(eMoverResult);

eSelectorState                        := f_GetState   (GVL_XTS.MoverSelectorState.State.State);
eSelectorResult                       := f_GetProgress(GVL_XTS.MoverSelectorState.State.State);

sSelectorState                        := TO_STRING(eSelectorState);
sSelectorResult                       := TO_STRING(eSelectorResult);

sStationState                         := TO_STRING(GVL_XTS.StationState[nStationSelected].State);
sStationStateMask                     := Tc2_Utilities.BYTE_TO_BINSTR(GVL_XTS.StationState[nStationSelected].nMask, 8);
sStationCtrlMask                      := Tc2_Utilities.BYTE_TO_BINSTR(GVL_XTS.StationCtrl[nStationSelected].nMask, 8);

tStationSelectedQueue                 := GVL_XTS.StationQueue[nStationSelected];
//############################################################################
//############################################################################
END_ACTION

END_PROGRAM

// ---- _XML/Configuration/fb_Configuration.TcPOU
//---------------------------------------------------------------------------------------------------------------
//
//  fb_Configuration
//
//  HAUD 2023.04.14
//  - base xml integration
//
//  HAUD 2026.04.10.
//  - now extending a base class
//
//  - cyclic OnChange wrapper for xml data 
//      - Ctrl/State
//        1. INIT
//        2. READ / WRITE
//
//  - read  ST_STATION_PARAMETER on demand
//  - write ST_STATION_PARAMETER on demand
//
//---------------------------------------------------------------------------------------------------------------
// This SOFTWARE is provided as an Example by THE PROVIDER "as is" and "with all faults." THE PROVIDER makes no 
// representations or warranties of any kind concerning the safety, suitability, lack of viruses, inaccuracies, 
// typographical errors, or other harmful components of this SOFTWARE. There are inherent dangers in the use of 
// any software, and you are solely responsible for determining whether this SOFTWARE is compatible with your 
// equipment and other software installed on your equipment. You are also solely responsible for the protection 
// of your equipment and backup of your data, and THE PROVIDER will not be liable for any damages you may suffer 
// in connection with using, modifying, or distributing this SOFTWARE.
//---------------------------------------------------------------------------------------------------------------
FUNCTION_BLOCK fb_Configuration EXTENDS fb_XmlBase
VAR
  _stCtrl               : REFERENCE TO ST_DATA_CTRL;
  _stState              : REFERENCE TO ST_DATA_STATE;

  _stConfiguration      : ST_Configuration;
  _pStationParameter    : POINTER TO ARRAY[1..MAX_STATION] OF ST_STATION_PARAMETER;
END_VAR
VAR CONSTANT
  FILE_ROOT             : STRING := 'CONFIG_XtsTransport_';
  X_PATH                : STRING := '/XtsTransport/config';
END_VAR

//---------------------------------------------------------------------------------------------------------------
//  check pointers from the outside
//---------------------------------------------------------------------------------------------------------------
IF NOT Check() THEN RETURN; END_IF
//---------------------------------------------------------------------------------------------------------------
// always build the internal data pointer
//  - as always: better safe than sorry
//  - leave this bit here, it doesn't cost much and safely addresses the data
//---------------------------------------------------------------------------------------------------------------
_pData                        := ADR    (_stConfiguration);
_nData                        := SIZEOF (_stConfiguration);
_sXpath                       := X_PATH;

// copy to local for debug
_eCmd                         := _stCtrl.Cmd;

// cyclic check for command change
// get state for cmd
IF (_eCmd <> _eCmdOld)
THEN
  // get matching sdtate for Ctrl.Cmd
  _eState                     := Cmd(_eCmd);
  _eCmdOld                    := _eCmd;
END_IF


CASE _eResult
OF
  E_PROGRESS.PROGRESS_INVALID:
    _stState.State            := E_DATA_STATE.NULL;

  E_PROGRESS.PROGRESS_ERROR:
    _stState.State            := _eState + E_PROGRESS.PROGRESS_ERROR;

  E_PROGRESS.PROGRESS_DONE:
    _stState.State            := _eState + E_PROGRESS.PROGRESS_DONE;

ELSE
  // work in progress
  // update progress for extern use
  _stState.State              := _eState + _eResult;

  CASE _eState
  OF
    E_DATA_STATE.INIT:
      _eResult   := _eInit    := CreateFolder(TRUE);

    E_DATA_STATE.READ:
      _eResult                := XmlRead(TRUE);
      IF (_eResult = E_PROGRESS.PROGRESS_DONE)
      THEN
        // copy the single ladies
        memcpy(_pStationParameter, ADR(_stConfiguration.XtsStationParameter), SIZEOF(_stConfiguration.XtsStationParameter));
      END_IF

    E_DATA_STATE.WRITE:
      _eResult                := XmlWrite(TRUE);
  ELSE
      _eResult                := E_PROGRESS.PROGRESS_INVALID;
  END_CASE
END_CASE

METHOD Check : BOOL
//-------------------------------------------------------------------------
IF NOT (__ISVALIDREF(_stCtrl))
THEN
  _eCheck               := E_DATA_CHECK.REFERENCE_CTRL_INVALID;
  RETURN;
END_IF
//-------------------------------------------------------------------------
IF NOT (__ISVALIDREF(_stState))
THEN
  _eCheck               := E_DATA_CHECK.REFERENCE_STATE_INVALID;
  RETURN;
END_IF
//-------------------------------------------------------------------------
IF NOT (_pStationParameter <> 0)
THEN
  _eCheck               := E_DATA_CHECK.POINTER_STATION_PARAMETER_INVALID;
  RETURN;
END_IF
//-------------------------------------------------------------------------
_eCheck                 := E_DATA_CHECK.DONE_CHECK;
Check                   := TRUE;
END_METHOD

METHOD PRIVATE Cmd : E_DATA_STATE
VAR_INPUT
  Ctrl      : E_DATA_CTRL;
END_VAR
VAR_INST
  _eState   : E_DATA_STATE;
END_VAR
IF NOT Check() THEN Cmd   := E_DATA_STATE.NULL;  RETURN; END_IF

CASE Ctrl
OF
  //---------------------------------------------------------------
  E_DATA_CTRL.INIT:
    _sName                := concat(FILE_ROOT, _sIdentity);
    _sName                := concat(_sName, '.xml');
    _sFilePath            := concat(_sDirectoryPath, _sName);

    _eInit                := E_PROGRESS.PROGRESS_INVALID;
    _eResult              := CreateFolder(FALSE);
    _eState               := E_DATA_STATE.INIT;
  //---------------------------------------------------------------
  E_DATA_CTRL.READ:
    _eResult              := XmlRead(FALSE);
    _eState               := E_DATA_STATE.READ;
  //---------------------------------------------------------------
  E_DATA_CTRL.WRITE:
    _stConfiguration.XtsStationParameter  := _pStationParameter^;

    _eResult              := XmlWrite(FALSE);
    _eState               := E_DATA_STATE.WRITE;
ELSE
  //---------------------------------------------------------------
    _eResult              := E_PROGRESS.PROGRESS_INVALID; 
    _eState               := E_DATA_STATE.NO_EXIST;
END_CASE

Cmd                       := _eState;
END_METHOD

PROPERTY Ctrl : REFERENCE to ST_DATA_CTRL
SET
_stCtrl ref= Ctrl;
END_SET
END_PROPERTY

PROPERTY Identity : OTCID
GET
Identity := _XpuIdentity;
END_GET
SET
_XpuIdentity  := Identity;
_sIdentity    := Tc2_Utilities.DWORD_TO_HEXSTR(_XpuIdentity,8,FALSE);
END_SET
END_PROPERTY

PROPERTY State : REFERENCE TO ST_DATA_STATE
SET
_stState ref= State;
END_SET
END_PROPERTY

PROPERTY StationParameter : pointer to ARRAY[1..MAX_STATION] OF ST_STATION_PARAMETER
SET
_pStationParameter := StationParameter;
END_SET
END_PROPERTY

END_FUNCTION_BLOCK

// ---- _XML/fb_XmlBase.TcPOU
//---------------------------------------------------------------------------------------------------------------
//
//  HAUD 2026.04.10.
//
//  fb_XmlBase
//    - wraps xml read
//    - wraps xml write
//
//   - abstract base class for extending xml R/W ctrl for any data
//
//---------------------------------------------------------------------------------------------------------------
// This SOFTWARE is provided as an Example by THE PROVIDER "as is" and "with all faults." THE PROVIDER makes no 
// representations or warranties of any kind concerning the safety, suitability, lack of viruses, inaccuracies, 
// typographical errors, or other harmful components of this SOFTWARE. There are inherent dangers in the use of 
// any software, and you are solely responsible for determining whether this SOFTWARE is compatible with your 
// equipment and other software installed on your equipment. You are also solely responsible for the protection 
// of your equipment and backup of your data, and THE PROVIDER will not be liable for any damages you may suffer 
// in connection with using, modifying, or distributing this SOFTWARE.
//---------------------------------------------------------------------------------------------------------------
FUNCTION_BLOCK ABSTRACT fb_XmlBase
VAR
  //------------------------------------------------------------------------------------------------------------
  // pointer check result
  //------------------------------------------------------------------------------------------------------------
  _eCheck                     : E_DATA_CHECK;
  _sCheck                     : STRING;
  //------------------------------------------------------------------------------------------------------------
  // internal control and state
  //------------------------------------------------------------------------------------------------------------
  _eInit                      : E_PROGRESS;
  _eCmd,
  _eCmdOld                    : E_DATA_CTRL;
  _eState                     : E_DATA_STATE;
  _eResult                    : E_PROGRESS;
  //------------------------------------------------------------------------------------------------------------
  // Tc2_XmlDataSrv wrappers
  //------------------------------------------------------------------------------------------------------------
  _fbXmlRead                  : fb_XmlRead;
  _fbXmlWrite                 : fb_XmlWrite;
  //------------------------------------------------------------------------------------------------------------
  // who am I?
  //  - Identity built in extending class
  //
  // see fb_Configuration.Identity.Set() as example
  //------------------------------------------------------------------------------------------------------------
  {attribute 'displaymode' := 'hex'}
  _XpuIdentity                : OTCID;        // identity must be set by extending class
  _sIdentity                  : STRING;       // part of filename
  //------------------------------------------------------------------------------------------------------------
  // where am I?
  //  - hocus pocus
  //    - you have to define my locus 
  //
  // see fb_Configuration.Identity.Set() as example
  //------------------------------------------------------------------------------------------------------------
  _sDirectoryPath             : STRING;       // root directory for data
  _sFilePath                  : STRING(255);  // path and filename (shall include identity in filepath)

  _sName                      : STRING;       // filename with *.xml
  _sXpath                     : STRING;       // XPath from extending class
  //------------------------------------------------------------------------------------------------------------
  // what am I?
  //  - data from the void
  //------------------------------------------------------------------------------------------------------------
  _pData                      : Global.PVOID;
  _nData                      : UDINT;
  //------------------------------------------------------------------------------------------------------------
  _eDeviceIdentifier          : e_Device;
  _stMsg                      : ST_Message;
  _eMessageLevel              : E_MessageType;
END_VAR

METHOD CreateFolder : E_PROGRESS
VAR_INPUT
  Execute         : BOOL;
END_VAR
VAR_INST
  _nErrorId       : UDINT;
  _eState         : E_PROGRESS;
  _sPath          : Tc2_System.T_MaxString;
  _fbCreateDir    : Tc2_System.FB_CreateDir;
END_VAR

IF NOT Execute
THEN
  _eState                     := E_PROGRESS.PROGRESS_INIT;
END_IF


CASE _eState
OF
  E_PROGRESS.PROGRESS_INIT:
    IF Execute
    THEN
      _eState                 := E_PROGRESS.PROGRESS_BUSY;
      _nErrorId               := 0;

      _fbCreateDir(
                    sNetId    := '', 
                    sPathName := _sPath, 
                    ePath     := Tc2_System.E_OpenPath.PATH_GENERIC, 
                    bExecute  := FALSE, 
                    tTimeout  := T#1S);
    END_IF

  E_PROGRESS.PROGRESS_BUSY:
    _fbCreateDir(
                  sNetId      := '', 
                  sPathName   := _sPath, 
                  ePath       := Tc2_System.E_OpenPath.PATH_GENERIC, 
                  bExecute    := TRUE, 
                  tTimeout    := T#1S,
                  nErrId      => _nErrorId);

    IF _fbCreateDir.bBusy
    THEN
      _eState                 := E_PROGRESS.PROGRESS_OCCUPIED;
    END_IF

  E_PROGRESS.PROGRESS_OCCUPIED:
    _fbCreateDir(
                  sNetId      := '', 
                  sPathName   := _sPath, 
                  ePath       := Tc2_System.E_OpenPath.PATH_GENERIC, 
                  bExecute    := TRUE, 
                  tTimeout    := T#1S,
                  nErrId      => _nErrorId);

    IF NOT _fbCreateDir.bBusy
    THEN
      _eState                 := E_PROGRESS.PROGRESS_WORKING;
    END_IF

  E_PROGRESS.PROGRESS_WORKING:
    _eState                   := E_PROGRESS.PROGRESS_DONE;
    _fbCreateDir(
                  sNetId      := '', 
                  sPathName   := _sPath, 
                  ePath       := Tc2_System.E_OpenPath.PATH_GENERIC, 
                  bExecute    := FALSE, 
                  tTimeout    := T#1S);

    IF (_eMessageLevel > E_MessageType.eMessageError)
    THEN
      _stMsg.eType            := E_MessageType.eMessageInfo;
      _stMsg.eDevice          := _eDeviceIdentifier;
      _stMsg.eSubdevice       := e_Subdevice.fbCreateFolder;
      _stMsg.iErrorNumber     := 0;
      _stMsg.sText            := concat(' : ', TO_STRING(_eState));
      f_MessageSet(_stMsg);
    END_IF
END_CASE

CreateFolder                  := _eState;
END_METHOD

PROPERTY FilePath : string(255)
GET
FilePath := _sFilePath;
END_GET
END_PROPERTY

PROPERTY FolderPath : string
GET
FolderPath := _sDirectoryPath;
END_GET
SET
_sDirectoryPath := FolderPath;
END_SET
END_PROPERTY

PROPERTY MessageDevice : udint
SET
_eDeviceIdentifier   := MessageDevice;
END_SET
END_PROPERTY

PROPERTY MessageLevel : e_messagetype
SET
_eMessageLevel := MessageLevel;
END_SET
END_PROPERTY

METHOD XmlRead  : E_PROGRESS
VAR_INPUT
  Execute               : BOOL;
END_VAR
VAR_INST
  _eState               : E_PROGRESS;
  _nErrorId             : UDINT;
END_VAR

IF NOT Execute
THEN
  _eState                     := E_PROGRESS.PROGRESS_INIT;
END_IF

CASE _eState
OF
  E_PROGRESS.PROGRESS_INIT:
    IF Execute
    THEN
      _nErrorId               := 0;
      _eState                 := E_PROGRESS.PROGRESS_BUSY;

      IF (_eMessageLevel > E_MessageType.eMessageInfo)
      THEN
        _stMsg.eType          := E_MessageType.eMessageVerbose;
        _stMsg.eDevice        := _eDeviceIdentifier;
        _stMsg.eSubdevice     := e_Subdevice.fbXmlRead;
        _stMsg.iErrorNumber   := _nErrorId;
        _stMsg.sText          := concat(' : ', TO_STRING(_eState));
        f_MessageSet(_stMsg);
      END_IF
    END_IF

  E_PROGRESS.PROGRESS_BUSY:
    _eState                   := E_PROGRESS.PROGRESS_OCCUPIED;
    _fbXmlRead(
              bExecute        := FALSE, 
              sFilePath       := _sFilePath, 
              sXPath          := _sXpath, 
              pData           := _pData, 
              diSize          := _nData);

  E_PROGRESS.PROGRESS_OCCUPIED:
    _fbXmlRead(
              bExecute        := TRUE);

    IF _fbXmlRead.bError
    THEN
      _nErrorId               := _fbXmlRead.nError;
      _eState                 := E_PROGRESS.PROGRESS_ERROR;

      _stMsg.eType            := E_MessageType.eMessageError;
      _stMsg.eDevice          := _eDeviceIdentifier;
      _stMsg.eSubdevice       := e_Subdevice.fbXmlRead;
      _stMsg.iErrorNumber     := _nErrorId;
      _stMsg.sText            := concat(' : ', TO_STRING(_eState));
      f_MessageSet(_stMsg);

      _fbXmlRead(
              bExecute        := FALSE);

    ELSIF _fbXmlRead.bDone
    THEN
      _eState                 := E_PROGRESS.PROGRESS_WORKING;
      _fbXmlRead(
              bExecute        := FALSE);
    END_IF

  E_PROGRESS.PROGRESS_WORKING:
    _eState                   := E_PROGRESS.PROGRESS_DONE;

    IF (_eMessageLevel > E_MessageType.eMessageError)
    THEN
      _stMsg.eType            := E_MessageType.eMessageInfo;
      _stMsg.eDevice          := _eDeviceIdentifier;
      _stMsg.eSubdevice       := e_Subdevice.fbXmlRead;
      _stMsg.iErrorNumber     := _nErrorId;
      _stMsg.sText            := concat(' : ', TO_STRING(_eState));
      f_MessageSet(_stMsg);
    END_IF
END_CASE

XmlRead                       := _eState;
END_METHOD

METHOD XmlWrite : E_PROGRESS
VAR_INPUT
  Execute               : BOOL;
END_VAR
VAR_INST
  _eState               : E_PROGRESS;
  _nErrorId             : UDINT;
END_VAR

IF NOT Execute
THEN
  _eState                     := E_PROGRESS.PROGRESS_INIT;
END_IF

CASE _eState
OF
  E_PROGRESS.PROGRESS_INIT:
    IF Execute
    THEN
      _nErrorId               := 0;
      _eState                 := E_PROGRESS.PROGRESS_BUSY;

      IF (_eMessageLevel > E_MessageType.eMessageInfo)
      THEN
        _stMsg.eType          := E_MessageType.eMessageVerbose;
        _stMsg.eDevice        := _eDeviceIdentifier;
        _stMsg.eSubdevice     := e_Subdevice.fbXmlWrite;
        _stMsg.iErrorNumber   := _nErrorId;
        _stMsg.sText          := concat(' : ', TO_STRING(_eState));
        f_MessageSet(_stMsg);
      END_IF
    END_IF

  E_PROGRESS.PROGRESS_BUSY:
    _eState                   := E_PROGRESS.PROGRESS_OCCUPIED;
    _fbXmlWrite(
              bExecute        := FALSE, 
              sFilePath       := _sFilePath, 
              sXPath          := _sXpath, 
              pData           := _pData, 
              diSize          := _nData);

  E_PROGRESS.PROGRESS_OCCUPIED:
    _fbXmlWrite(
              bExecute        := TRUE);

    IF _fbXmlWrite.bError
    THEN
      _nErrorId               := _fbXmlRead.nError;
      _eState                 := E_PROGRESS.PROGRESS_ERROR;

      _stMsg.eType            := E_MessageType.eMessageError;
      _stMsg.eDevice          := _eDeviceIdentifier;
      _stMsg.eSubdevice       := e_Subdevice.fbXmlWrite;
      _stMsg.iErrorNumber     := _nErrorId;
      _stMsg.sText            := concat(' : ', TO_STRING(_eState));
      f_MessageSet(_stMsg);

      _fbXmlWrite(
              bExecute        := FALSE);

    ELSIF _fbXmlWrite.bDone
    THEN
      _eState                 := E_PROGRESS.PROGRESS_WORKING;
      _fbXmlWrite(
              bExecute        := FALSE);
    END_IF

  E_PROGRESS.PROGRESS_WORKING:
    _eState                   := E_PROGRESS.PROGRESS_DONE;

    IF (_eMessageLevel > E_MessageType.eMessageError)
    THEN
      _stMsg.eType            := E_MessageType.eMessageInfo;
      _stMsg.eDevice          := _eDeviceIdentifier;
      _stMsg.eSubdevice       := e_Subdevice.fbXmlWrite;
      _stMsg.iErrorNumber     := _nErrorId;
      _stMsg.sText            := concat(' : ', TO_STRING(_eState));
      f_MessageSet(_stMsg);
    END_IF
END_CASE

XmlWrite                      := _eState;
END_METHOD

END_FUNCTION_BLOCK

// ---- _XML/PositionOffsets/fb_MoverPositionOffsetData.TcPOU
//---------------------------------------------------------------------------------------------------------------
//
//  fb_MoverPositionOffsetData
//
//  HAUD 2026.05.08.
//  - xml handler for Position offsets of the movers in stations
//
//  - cyclic OnChange wrapper for xml data 
//      - Ctrl/State
//        1. INIT
//        2. READ / WRITE
//
//  - read  ST_MOVER_OFFSETS on demand
//  - write ST_MOVER_OFFSETS on demand
//
//---------------------------------------------------------------------------------------------------------------
// This SOFTWARE is provided as an Example by THE PROVIDER "as is" and "with all faults." THE PROVIDER makes no 
// representations or warranties of any kind concerning the safety, suitability, lack of viruses, inaccuracies, 
// typographical errors, or other harmful components of this SOFTWARE. There are inherent dangers in the use of 
// any software, and you are solely responsible for determining whether this SOFTWARE is compatible with your 
// equipment and other software installed on your equipment. You are also solely responsible for the protection 
// of your equipment and backup of your data, and THE PROVIDER will not be liable for any damages you may suffer 
// in connection with using, modifying, or distributing this SOFTWARE.
//---------------------------------------------------------------------------------------------------------------
FUNCTION_BLOCK fb_MoverPositionOffsetData EXTENDS fb_XmlBase
VAR
  _stCtrl               : REFERENCE TO ST_DATA_CTRL;
  _stState              : REFERENCE TO ST_DATA_STATE;

  _stData               : ST_MOVER_OFFSETS;
  _pPositionOffset      : POINTER TO ARRAY[1..MAX_STATION] OF T_NEST_OFFSET; // added to PosStop[] in XtsStation
END_VAR
VAR CONSTANT
  FILE_ROOT             : STRING := 'OFFSET_XtsTransport_';
  X_PATH                : STRING := '/XtsTransport/PositionOffset';
END_VAR

//---------------------------------------------------------------------------------------------------------------
//  check pointers from the outside
//---------------------------------------------------------------------------------------------------------------
IF NOT Check() THEN RETURN; END_IF
//---------------------------------------------------------------------------------------------------------------
// always build the internal data pointer
//  - as always: better safe than sorry
//  - leave this bit here, it doesn't cost much and safely addresses the data
//---------------------------------------------------------------------------------------------------------------
_pData                        := ADR    (_stData);
_nData                        := SIZEOF (_stData);
_sXpath                       := X_PATH;

// copy to local for debug
_eCmd                         := _stCtrl.Cmd;

// cyclic check for command change
// get state for cmd
IF (_eCmd <> _eCmdOld)
THEN
  // get matching sdtate for Ctrl.Cmd
  _eState                     := Cmd(_eCmd);
  _eCmdOld                    := _eCmd;
END_IF


CASE _eResult
OF
  E_PROGRESS.PROGRESS_INVALID:
    _stState.State            := E_DATA_STATE.NULL;

  E_PROGRESS.PROGRESS_ERROR:
    _stState.State            := _eState + E_PROGRESS.PROGRESS_ERROR;

  E_PROGRESS.PROGRESS_DONE:
    _stState.State            := _eState + E_PROGRESS.PROGRESS_DONE;

ELSE
  // work in progress
  // update progress for extern use
  _stState.State              := _eState + _eResult;

  CASE _eState
  OF
    E_DATA_STATE.INIT:
      _eResult   := _eInit    := CreateFolder(TRUE);

    E_DATA_STATE.READ:
      _eResult                := XmlRead(TRUE);
      IF (_eResult = E_PROGRESS.PROGRESS_DONE)
      THEN
        // copy the single ladies
        memcpy(_pPositionOffset, ADR(_stData.PositionOffset), SIZEOF(_stData.PositionOffset));
      END_IF

    E_DATA_STATE.WRITE:
      _eResult                := XmlWrite(TRUE);
  ELSE
      _eResult                := E_PROGRESS.PROGRESS_INVALID;
  END_CASE
END_CASE

METHOD Check : BOOL
//-------------------------------------------------------------------------
IF NOT (__ISVALIDREF(_stCtrl))
THEN
  _eCheck               := E_DATA_CHECK.REFERENCE_CTRL_INVALID;
  RETURN;
END_IF
//-------------------------------------------------------------------------
IF NOT (__ISVALIDREF(_stState))
THEN
  _eCheck               := E_DATA_CHECK.REFERENCE_STATE_INVALID;
  RETURN;
END_IF
//-------------------------------------------------------------------------
IF NOT (_pPositionOffset <> 0)
THEN
  _eCheck               := E_DATA_CHECK.POINTER_MOVER_OFFSETS_INVALID;
  RETURN;
END_IF
//-------------------------------------------------------------------------
_eCheck                 := E_DATA_CHECK.DONE_CHECK;
Check                   := TRUE;
END_METHOD

METHOD PRIVATE Cmd : E_DATA_STATE
VAR_INPUT
  Ctrl      : E_DATA_CTRL;
END_VAR
VAR_INST
  _eState   : E_DATA_STATE;
END_VAR
IF NOT Check() THEN Cmd   := E_DATA_STATE.NULL;  RETURN; END_IF

CASE Ctrl
OF
  //---------------------------------------------------------------
  E_DATA_CTRL.INIT:
    _sName                := concat(FILE_ROOT, _sIdentity);
    _sName                := concat(_sName, '.xml');
    _sFilePath            := concat(_sDirectoryPath, _sName);

    _eInit                := E_PROGRESS.PROGRESS_INVALID;
    _eResult              := CreateFolder(FALSE);
    _eState               := E_DATA_STATE.INIT;
  //---------------------------------------------------------------
  E_DATA_CTRL.READ:
    _eResult              := XmlRead(FALSE);
    _eState               := E_DATA_STATE.READ;
  //---------------------------------------------------------------
  E_DATA_CTRL.WRITE:
    _stData.PositionOffset  := _pPositionOffset^;

    _eResult              := XmlWrite(FALSE);
    _eState               := E_DATA_STATE.WRITE;
ELSE
  //---------------------------------------------------------------
    _eResult              := E_PROGRESS.PROGRESS_INVALID; 
    _eState               := E_DATA_STATE.NO_EXIST;
END_CASE

Cmd                       := _eState;
END_METHOD

PROPERTY Ctrl : REFERENCE to ST_DATA_CTRL
SET
_stCtrl ref= Ctrl;
END_SET
END_PROPERTY

PROPERTY Identity : OTCID
GET
Identity := _XpuIdentity;
END_GET
SET
_XpuIdentity  := Identity;
_sIdentity    := Tc2_Utilities.DWORD_TO_HEXSTR(_XpuIdentity,8,FALSE);
END_SET
END_PROPERTY

PROPERTY MoverOffsets : pointer to ARRAY[1..MAX_STATION] OF T_NEST_OFFSET
SET
_pPositionOffset := MoverOffsets;
END_SET
END_PROPERTY

PROPERTY State : REFERENCE TO ST_DATA_STATE
SET
_stState ref= State;
END_SET
END_PROPERTY

END_FUNCTION_BLOCK

// ---- APPLICATION/XTS_TRANSPORT_1.TcVIS
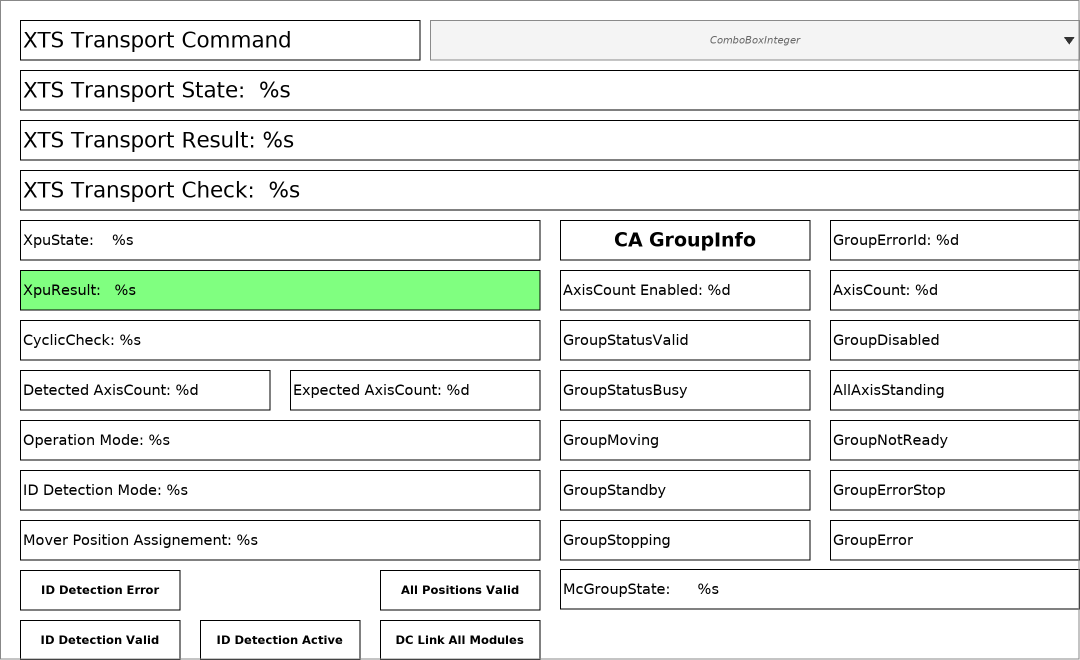
VISUALIZATION XTS_TRANSPORT_1  // 1080x660
    Rectangle (20,20 400x40), "XTS Transport Command"
    ComboBoxInteger (430,20 650x40), variable: GVL_XTS.XtsTransportCtrl.Cmd, text list: 'TL_E_CTRL_TRANSPORT'
    Rectangle (20,70 1060x40), "XTS Transport State: %s", text variable: MAIN.sTransportState
    Rectangle (20,120 1060x40), "XTS Transport Result: %s", text variable: MAIN.sTransportResult
    Rectangle (20,170 1060x40), "XTS Transport Check: %s", text variable: MAIN.sTransportCheck
    Frame (20,220 520x440)
        shows XPU_VISU(stXpuState := GVL_XTS.XtsTransportState.XpuState, stXpuInfo := GVL_XTS.XtsTransportState.XpuInfo, stXpuStrings := MAIN.stXpuStrings)
    Frame (560,220 520x390)
        shows GROUP_VISU(stGroupInfo := GVL_XTS.XtsTransportState.GroupInfo, sGroupState := MAIN.sCaGroupState)
END_VISUALIZATION

// ---- XTS_TRANSPORT/_Visualization/GROUP_VISU.TcVIS
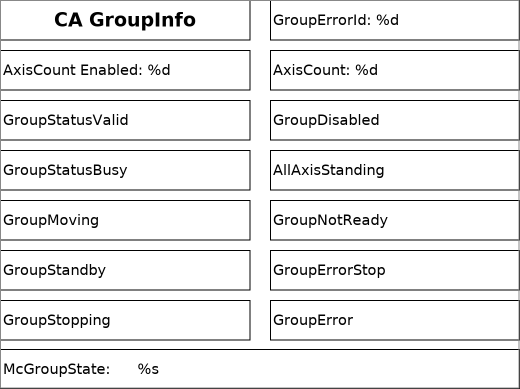
VISUALIZATION GROUP_VISU  // 520x389
VAR_IN_OUT
	stGroupInfo   : ST_GROUP_INFO;
  sGroupState   : string(60);
END_VAR
    Rectangle (0,100 250x40), "GroupStatusValid", colour toggle: stGroupInfo.GroupStatusValid
    Rectangle (0,150 250x40), "GroupStatusBusy", colour toggle: stGroupInfo.GroupStatusBusy
    Rectangle (0,200 250x40), "GroupMoving", colour toggle: stGroupInfo.GroupMoving
    Rectangle (270,250 250x40), "GroupErrorStop", colour toggle: stGroupInfo.GroupErrorStop
    Rectangle (270,200 250x40), "GroupNotReady", colour toggle: stGroupInfo.GroupNotReady
    Rectangle (0,250 250x40), "GroupStandby", colour toggle: stGroupInfo.GroupStandby
    Rectangle (0,300 250x40), "GroupStopping", colour toggle: stGroupInfo.GroupStopping
    Rectangle (270,100 250x40), "GroupDisabled", colour toggle: stGroupInfo.GroupDisabled
    Rectangle (270,150 250x40), "AllAxisStanding", colour toggle: stGroupInfo.AllAxesStanding
    Rectangle (270,300 250x40), "GroupError", colour toggle: stGroupInfo.GroupError
    Rectangle (270,0 250x40), "GroupErrorId: %d", text variable: stGroupInfo.GroupErrorId
    Rectangle (270,50 250x40), "AxisCount: %d", text variable: stGroupInfo.AxisCount
    Rectangle (0,349 520x40), "McGroupState: %s", text variable: sGroupState
    Rectangle (0,0 250x40), "CA GroupInfo"
    Rectangle (0,50 250x40), "AxisCount Enabled: %d", text variable: stGroupInfo.AxisCountEnabled
END_VISUALIZATION

// ---- XTS_TRANSPORT/_Visualization/MOVER_VISU.TcVIS
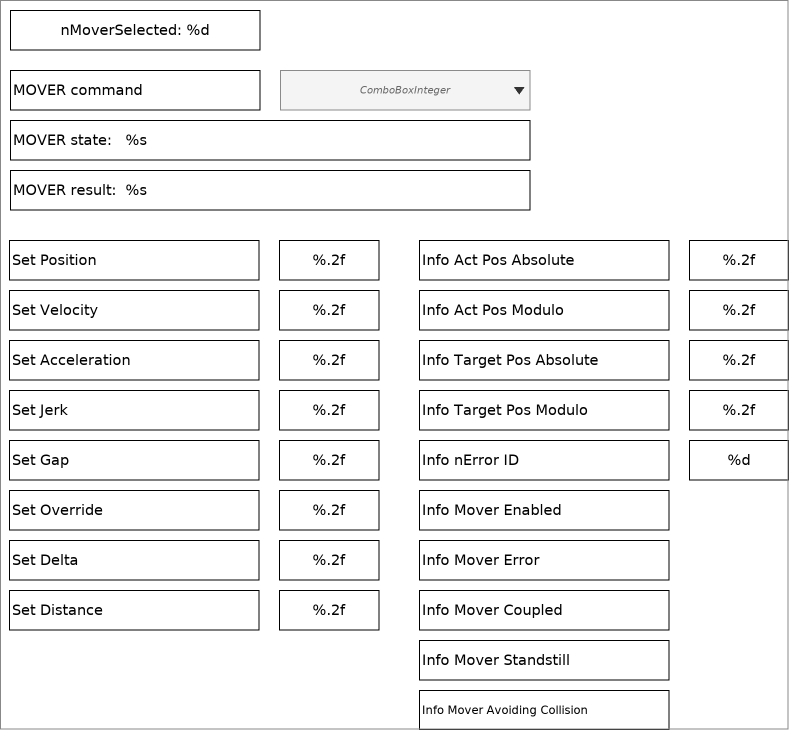
VISUALIZATION MOVER_VISU  // 789x730
    Rectangle (10,10 250x40), "nMoverSelected: %d", text variable: MAIN.nMoverSelected
        OnMouseClick: write the text variable via VisuDialogs.Numpad, min 1, max MAX_MOVER, title 'Selected Mover'
    Rectangle (10,120 520x40), "MOVER state: %s", text variable: MAIN.sMoverState
    Rectangle (10,70 250x40), "MOVER command"
    ComboBoxInteger (280,70 250x40), variable: GVL_XTS.MoverCtrl[MAIN.nMoverSelected].Cmd, text list: 'TL_E_CTRL_MOVER'
    Rectangle (10,170 520x40), "MOVER result: %s", text variable: MAIN.sMoverResult
    Rectangle (9,240 250x40), "Set Position"
    Rectangle (9,290 250x40), "Set Velocity"
    Rectangle (9,340 250x40), "Set Acceleration"
    Rectangle (9,390 250x40), "Set Jerk"
    Rectangle (9,440 250x40), "Set Gap"
    Rectangle (9,490 250x40), "Set Override"
    Rectangle (9,540 250x40), "Set Delta"
    Rectangle (9,590 250x40), "Set Distance"
    Rectangle (279,240 100x40), "%.2f", text variable: GVL_XTS.MoveData[MAIN.nMoverSelected].rPos
        OnMouseClick: write the text variable via Default
    Rectangle (279,290 100x40), "%.2f", text variable: GVL_XTS.MoveData[MAIN.nMoverSelected].rVelo
        OnMouseClick: write the text variable via Default
    Rectangle (279,340 100x40), "%.2f", text variable: GVL_XTS.MoveData[MAIN.nMoverSelected].rAcc
        OnMouseClick: write the text variable via Default
    Rectangle (279,390 100x40), "%.2f", text variable: GVL_XTS.MoveData[MAIN.nMoverSelected].rJerk
        OnMouseClick: write the text variable via Default
    Rectangle (279,440 100x40), "%.2f", text variable: GVL_XTS.MoveData[MAIN.nMoverSelected].rGap
        OnMouseClick: write the text variable via Default
    Rectangle (279,490 100x40), "%.2f", text variable: GVL_XTS.MoveData[MAIN.nMoverSelected].rOverride
        OnMouseClick: write the text variable via Default
    Rectangle (279,540 100x40), "%.2f", text variable: GVL_XTS.MoveData[MAIN.nMoverSelected].rDelta
        OnMouseClick: write the text variable via Default
    Rectangle (279,590 100x40), "%.2f", text variable: GVL_XTS.MoveData[MAIN.nMoverSelected].rDistance
        OnMouseClick: write the text variable via Default
    Rectangle (419,240 250x40), "Info Act Pos Absolute"
    Rectangle (419,290 250x40), "Info Act Pos Modulo"
    Rectangle (419,340 250x40), "Info Target Pos Absolute"
    Rectangle (419,390 250x40), "Info Target Pos Modulo"
    Rectangle (419,440 250x40), "Info nError ID"
    Rectangle (689,240 100x40), "%.2f", text variable: GVL_XTS.MoverInfo[MAIN.nMoverSelected].rAbsActPos
    Rectangle (689,290 100x40), "%.2f", text variable: GVL_XTS.MoverInfo[MAIN.nMoverSelected].rModuloActPos
    Rectangle (689,340 100x40), "%.2f", text variable: GVL_XTS.MoverInfo[MAIN.nMoverSelected].rAbsTargetPos
    Rectangle (689,390 100x40), "%.2f", text variable: GVL_XTS.MoverInfo[MAIN.nMoverSelected].rModuloTargetPos
    Rectangle (689,440 100x40), "%d", text variable: GVL_XTS.MoverInfo[MAIN.nMoverSelected].nErrorId
    Rectangle (419,490 250x40), "Info Mover Enabled", colour toggle: GVL_XTS.MoverInfo[MAIN.nMoverSelected].bMoverEnabled
    Rectangle (419,540 250x40), "Info Mover Error", colour toggle: GVL_XTS.MoverInfo[MAIN.nMoverSelected].bMoverError
    Rectangle (419,590 250x40), "Info Mover Coupled", colour toggle: GVL_XTS.MoverInfo[MAIN.nMoverSelected].bMoverCoupled
    Rectangle (419,640 250x40), "Info Mover Standstill", colour toggle: GVL_XTS.MoverInfo[MAIN.nMoverSelected].bMoverStandstill
    Rectangle (419,690 250x40), "Info Mover Avoiding Collision", colour toggle: GVL_XTS.MoverInfo[MAIN.nMoverSelected].bMoverAvoidingCollision
END_VISUALIZATION

// ---- XTS_TRANSPORT/_Visualization/SELECTOR_VISU.TcVIS
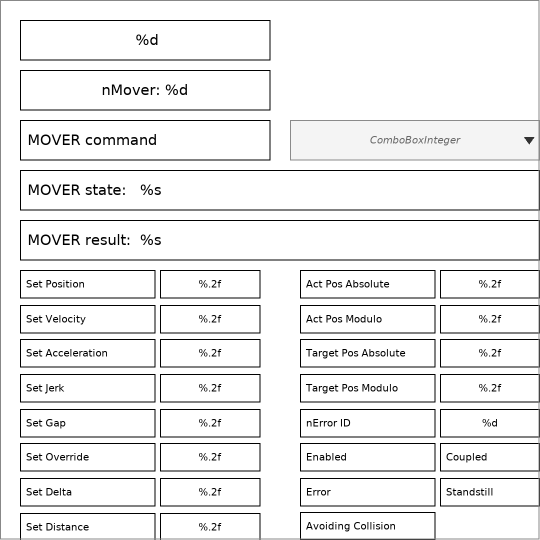
VISUALIZATION SELECTOR_VISU  // 540x540
    Frame (10,10 530x530)
        shows T_MOVER_SELECTOR(Control := GVL_XTS.SelectorCtrl, State := GVL_XTS.SelectorState, sState := MAIN.sSelectorState, sResult := MAIN.sSelectorResult)
END_VISUALIZATION

// ---- XTS_TRANSPORT/_Visualization/STATION_VISU.TcVIS
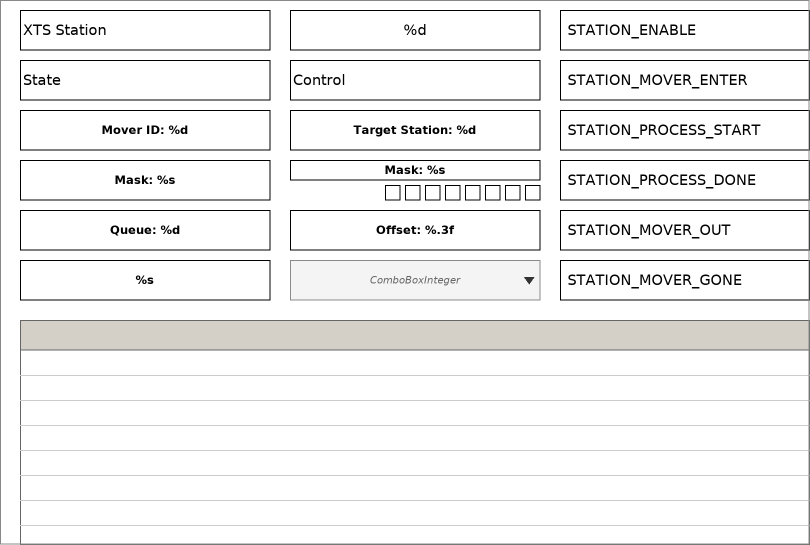
VISUALIZATION STATION_VISU  // 810x545
    Rectangle (20,10 250x40), "XTS Station"
    Rectangle (290,10 250x40), "%d", text variable: MAIN.nStationSelected
        OnMouseClick: write the text variable via VisuDialogs.Numpad, min 1, max MAX_STATION, title 'Selected Station'
    Rectangle (20,60 250x40), "State"
    Rectangle (290,60 250x40), "Control"
    Rectangle (20,210 250x40), "Queue: %d", text variable: GVL_XTS.StationState[MAIN.nStationSelected].nQueue
    Rectangle (20,110 250x40), "Mover ID: %d", text variable: GVL_XTS.StationState[MAIN.nStationSelected].nMoverId
    Rectangle (20,160 250x40), "Mask: %s", text variable: MAIN.sStationStateMask
    Rectangle (20,260 250x40), "%s", text variable: MAIN.sStationState
    ComboBoxInteger (290,260 250x40), variable: GVL_XTS.StationCtrl[MAIN.nStationSelected].eCmd, text list: 'TL_E_CTRL_STATION'
    Rectangle (290,210 250x40), "Offset: %.3f", text variable: GVL_XTS.StationCtrl[MAIN.nStationSelected].rOffset
    Rectangle (290,110 250x40), "Target Station: %d", text variable: GVL_XTS.StationCtrl[MAIN.nStationSelected].nTargetStation
        OnMouseClick: write the text variable via VisuDialogs.Numpad, min 1, max MAX_STATION, title 'Target Station'
    Rectangle (290,160 250x20), "Mask: %s", text variable: MAIN.sStationCtrlMask
    Rectangle (525,185 15x15)
        toggle GVL_XTS.StationCtrl[MAIN.nStationSelected].nMask.0
    Rectangle (505,185 15x15)
        toggle GVL_XTS.StationCtrl[MAIN.nStationSelected].nMask.1
    Rectangle (485,185 15x15)
        toggle GVL_XTS.StationCtrl[MAIN.nStationSelected].nMask.2
    Rectangle (465,185 15x15)
        toggle GVL_XTS.StationCtrl[MAIN.nStationSelected].nMask.3
    Rectangle (445,185 15x15)
        toggle GVL_XTS.StationCtrl[MAIN.nStationSelected].nMask.4
    Rectangle (425,185 15x15)
        toggle GVL_XTS.StationCtrl[MAIN.nStationSelected].nMask.5
    Rectangle (405,185 15x15)
        toggle GVL_XTS.StationCtrl[MAIN.nStationSelected].nMask.6
    Rectangle (385,185 15x15)
        toggle GVL_XTS.StationCtrl[MAIN.nStationSelected].nMask.7
    Rectangle (560,10 250x40), "STATION_ENABLE", colour toggle: MAIN.bStationEnable
        OnMouseClick: execute { GVL_XTS.StationCtrl[MAIN.nStationSelected].eCmd := E_STATION_CTRL.STATION_ENABLE; }
    Rectangle (560,60 250x40), "STATION_MOVER_ENTER", colour toggle: MAIN.bStationEnter
        OnMouseClick: execute { GVL_XTS.StationCtrl[MAIN.nStationSelected].eCmd := E_STATION_CTRL.STATION_MOVER_ENTER; }
    Rectangle (560,110 250x40), "STATION_PROCESS_START", colour toggle: MAIN.bStationStart
        OnMouseClick: execute { GVL_XTS.StationCtrl[MAIN.nStationSelected].eCmd := E_STATION_CTRL.STATION_PROCESS_START; }
    Rectangle (560,160 250x40), "STATION_PROCESS_DONE", colour toggle: MAIN.bStationDone
        OnMouseClick: execute { GVL_XTS.StationCtrl[MAIN.nStationSelected].eCmd := E_STATION_CTRL.STATION_PROCESS_DONE; }
    Rectangle (560,210 250x40), "STATION_MOVER_OUT", colour toggle: MAIN.bStationOut
        OnMouseClick: execute { GVL_XTS.StationCtrl[MAIN.nStationSelected].eCmd := E_STATION_CTRL.STATION_MOVER_OUT; }
    Rectangle (560,260 250x40), "STATION_MOVER_GONE", colour toggle: MAIN.bStationGone
        OnMouseClick: execute { GVL_XTS.StationCtrl[MAIN.nStationSelected].eCmd := E_STATION_CTRL.STATION_MOVER_GONE; }
    Table (20,320 790x225), data array: MAIN.tStationSelectedQueue
        p3854506369: MAIN.tStationSelectedQueue[INDEX].nMoverId
        p1892666644: MAIN.tStationSelectedQueue[INDEX].nTargetStation
        p338671338: MAIN.tStationSelectedQueue[INDEX].nMask
        p2170511999: MAIN.tStationSelectedQueue[INDEX].rOffset
END_VISUALIZATION

// ---- XTS_TRANSPORT/_Visualization/types/T_MOVER_SELECTOR.TcVIS
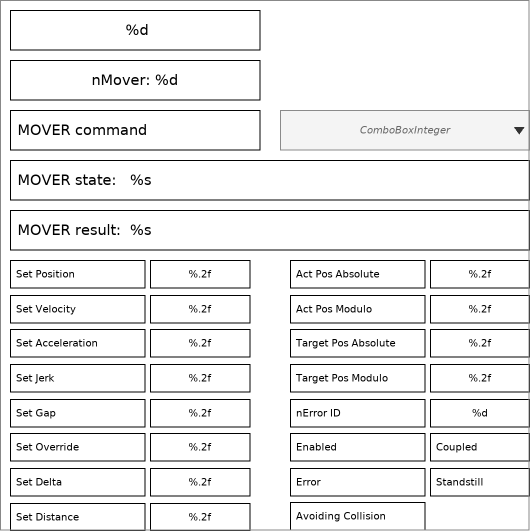
VISUALIZATION T_MOVER_SELECTOR  // 530x531
VAR_IN_OUT
	Control     : ST_MOVER_SELECTOR_CTRL;
  State       : ST_MOVER_SELECTOR_STATE;
  sState      : STRING;
  sResult     : STRING;
END_VAR
    Rectangle (10,60 250x40), "nMover: %d", text variable: Control.Mover
        OnMouseClick: write the text variable via VisuDialogs.Numpad, min 1, max MAX_MOVER, title 'Selected Mover'
    Rectangle (10,10 250x40), "%d", text variable: Control.Selector, text list: 'TL_E_MOVER_SELECTOR'
        OnMouseClick: write the text variable via VisuDialogs.Numpad, min 1, max MAX_MOVER, title 'Selected Mover'
    Rectangle (10,160 520x40), "MOVER state: %s", text variable: sState
    Rectangle (10,110 250x40), "MOVER command"
    ComboBoxInteger (280,110 250x40), variable: Control.Control.Cmd, text list: 'TL_E_CTRL_MOVER'
    Rectangle (10,210 520x40), "MOVER result: %s", text variable: sResult
    Rectangle (10,260 135x28), "Set Position"
    Rectangle (10,295 135x28), "Set Velocity"
    Rectangle (10,329 135x28), "Set Acceleration"
    Rectangle (10,364 135x28), "Set Jerk"
    Rectangle (10,399 135x28), "Set Gap"
    Rectangle (10,433 135x28), "Set Override"
    Rectangle (10,468 135x28), "Set Delta"
    Rectangle (10,503 135x28), "Set Distance"
    Rectangle (150,260 100x28), "%.2f", text variable: Control.Data.rPos
        OnMouseClick: write the text variable via Default
    Rectangle (150,295 100x28), "%.2f", text variable: Control.Data.rVelo
        OnMouseClick: write the text variable via Default
    Rectangle (150,329 100x28), "%.2f", text variable: Control.Data.rAcc
        OnMouseClick: write the text variable via Default
    Rectangle (150,364 100x28), "%.2f", text variable: Control.Data.rJerk
        OnMouseClick: write the text variable via Default
    Rectangle (150,399 100x28), "%.2f", text variable: Control.Data.rGap
        OnMouseClick: write the text variable via Default
    Rectangle (150,433 100x28), "%.2f", text variable: Control.Data.rOverride
        OnMouseClick: write the text variable via Default
    Rectangle (150,468 100x28), "%.2f", text variable: Control.Data.rDelta
        OnMouseClick: write the text variable via Default
    Rectangle (150,503 100x28), "%.2f", text variable: Control.Data.rDistance
        OnMouseClick: write the text variable via Default
    Rectangle (290,260 135x28), "Act Pos Absolute"
    Rectangle (290,295 135x28), "Act Pos Modulo"
    Rectangle (290,329 135x28), "Target Pos Absolute"
    Rectangle (290,364 135x28), "Target Pos Modulo"
    Rectangle (290,399 135x28), "nError ID"
    Rectangle (430,260 100x28), "%.2f", text variable: GVL_XTS.MoverInfo[MAIN.nMoverSelected].rAbsActPos
    Rectangle (430,295 100x28), "%.2f", text variable: GVL_XTS.MoverInfo[MAIN.nMoverSelected].rModuloActPos
    Rectangle (430,329 100x28), "%.2f", text variable: GVL_XTS.MoverInfo[MAIN.nMoverSelected].rAbsTargetPos
    Rectangle (430,364 100x28), "%.2f", text variable: GVL_XTS.MoverInfo[MAIN.nMoverSelected].rModuloTargetPos
    Rectangle (430,399 100x28), "%d", text variable: GVL_XTS.MoverInfo[MAIN.nMoverSelected].nErrorId
    Rectangle (290,433 135x28), "Enabled", colour toggle: GVL_XTS.MoverInfo[MAIN.nMoverSelected].bMoverEnabled
    Rectangle (290,468 135x28), "Error", colour toggle: GVL_XTS.MoverInfo[MAIN.nMoverSelected].bMoverError
    Rectangle (430,433 100x28), "Coupled", colour toggle: GVL_XTS.MoverInfo[MAIN.nMoverSelected].bMoverCoupled
    Rectangle (430,468 100x28), "Standstill", colour toggle: GVL_XTS.MoverInfo[MAIN.nMoverSelected].bMoverStandstill
    Rectangle (290,502 135x28), "Avoiding Collision", colour toggle: GVL_XTS.MoverInfo[MAIN.nMoverSelected].bMoverAvoidingCollision
END_VISUALIZATION

// ---- XTS_TRANSPORT/_Visualization/XPU_VISU.TcVIS
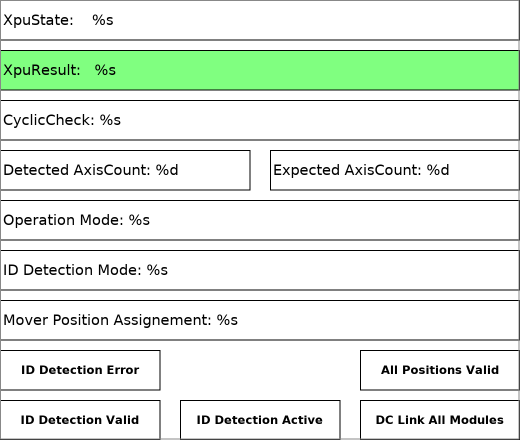
VISUALIZATION XPU_VISU  // 520x440
VAR_IN_OUT
	stXpuState    : ST_XPU_STATE;
  stXpuInfo     : ST_XPU_INFO;
  stXpuStrings  : ST_XPU_STRINGS;
END_VAR
    Rectangle (0,100 520x40), "CyclicCheck: %s", text variable: stXpuStrings.sXpuCyclicCheck
    Rectangle (0,0 520x40), "XpuState: %s", text variable: stXpuStrings.sXpuState
    Rectangle (0,50 520x40), "XpuResult: %s", text variable: stXpuStrings.sXpuResult, colour toggle: (MAIN.eXpuResult = E_PROGRESS.PROGRESS_ERROR)
    Rectangle (360,350 160x40), "All Positions Valid", colour toggle: stXpuInfo.AllPositionsValid
    Rectangle (0,350 160x40), "ID Detection Error", colour toggle: stXpuInfo.IdDetectionError
    Rectangle (0,400 160x40), "ID Detection Valid", colour toggle: stXpuInfo.IdDetectionValid
    Rectangle (180,400 160x40), "ID Detection Active", colour toggle: stXpuInfo.IdDetectionActive
    Rectangle (0,200 520x40), "Operation Mode: %s", text variable: stXpuStrings.sXpuOpMode
    Rectangle (0,250 520x40), "ID Detection Mode: %s", text variable: stXpuStrings.sXpuMoverId_DetectionMode
    Rectangle (0,300 520x40), "Mover Position Assignement: %s", text variable: stXpuStrings.sXpuMoverPosAssignement
    Rectangle (270,150 250x40), "Expected AxisCount: %d", text variable: stXpuInfo.nExpectedAxisCount
    Rectangle (0,150 250x40), "Detected AxisCount: %d", text variable: stXpuInfo.nDetectedAxisCount
    Rectangle (360,400 160x40), "DC Link All Modules", colour toggle: stXpuState.DcLink
END_VISUALIZATION
